// SIMATIC STEP 7 (V5.x) project Post-Platform V2
// CPU: CPU 313
// CPU: CPU 312IFM
// station: Hardware
// station: Master
// station: Hardware
// station: Slave
// station: P_ADR_BUS
// station: P_ADR_BUS
// station: P_ADR_BUS
// station: Configuration
// program: S7 Program(1)
// program: S7 Program(2)

SYMBOL_TABLE
"Counter.Balk"	C 0	COUNTER
"Geheugen.Platform"	DB 1	DB 1
"Geheugen.Instellingen"	DB 2	DB 2
"Uitgangen.Sturen"	FC 1	FC 1
"Merkers.Sturen"	FC 2	FC 2
"Timers + Counters"	FC 3	FC 3
"Berekeningen"	FC 4	FC 4
"Grafcet"	FC 5	FC 5
"Simulatie"	FC 6	FC 6
"Watch.Dog"	FC 7	FC 7
"Sub.Basis"	FC 14	FC 14
"Sub.Keuze"	FC 15	FC 15
"Sub.Keuze.Sta.A.or.B"	FC 16	FC 16
"Stap 0.0"	M 0.0	BOOL
"Stap 0.1"	M 0.1	BOOL
"Stap 0.2"	M 0.2	BOOL
"Stap 0.3"	M 0.3	BOOL
"Stap 0.4"	M 0.4	BOOL
"Stap 0.5"	M 0.5	BOOL
"Stap 0.6"	M 0.6	BOOL
"Stap 0.7"	M 0.7	BOOL
"Stap 1.0"	M 1.0	BOOL
"Stap 1.1"	M 1.1	BOOL
"Stap 1.2"	M 1.2	BOOL
"Stap 1.3"	M 1.3	BOOL
"Stap 1.4"	M 1.4	BOOL
"Stap 1.5"	M 1.5	BOOL
"Stap 1.6"	M 1.6	BOOL
"Stap 1.7"	M 1.7	BOOL
"Stap 2.0"	M 2.0	BOOL
"Stap 2.1"	M 2.1	BOOL
"Stap 2.2"	M 2.2	BOOL
"Stap 2.3"	M 2.3	BOOL
"Stap 2.4"	M 2.4	BOOL
"Stap 2.5"	M 2.5	BOOL
"Stap 2.6"	M 2.6	BOOL
"Stap 2.7"	M 2.7	BOOL
"Stap 3.0"	M 3.0	BOOL
"Stap 3.1"	M 3.1	BOOL
"Stap 3.2"	M 3.2	BOOL
"Stap 3.3"	M 3.3	BOOL
"Stap 3.4"	M 3.4	BOOL
"Stap 3.5"	M 3.5	BOOL
"Stap 3.6"	M 3.6	BOOL
"Stap 3.7"	M 3.7	BOOL
"Stap 4.0"	M 4.0	BOOL
"Stap 4.1"	M 4.1	BOOL
"Stap 4.2"	M 4.2	BOOL
"Stap 4.3"	M 4.3	BOOL
"Stap 4.4"	M 4.4	BOOL
"Stap 4.5"	M 4.5	BOOL
"Stap 4.6"	M 4.6	BOOL
"Stap 4.7"	M 4.7	BOOL
"Stop.Hardware"	M 10.0	BOOL
"Start.Hardware"	M 10.1	BOOL
"Sens.Sta.A.In"	M 10.2	BOOL
"Sens.Sta.A.Forward"	M 10.3	BOOL
"Sens.Sta.A.Down"	M 10.4	BOOL
"Sens.Sta.A.Up"	M 10.5	BOOL
"Sens.Sta.B.In"	M 10.6	BOOL
"Sens.Sta.B.Forward"	M 10.7	BOOL
"Sens.Sta.B.Down"	M 11.0	BOOL
"Sens.Sta.B.Up"	M 11.1	BOOL
"Sens.Proxi.1"	M 11.2	BOOL
"Sens.Proxi.2"	M 11.3	BOOL
"NoodStop.Relais"	M 11.4	BOOL
"Leeg"	M 12.0	BOOL
"Motor.Platform.Rechts"	M 12.1	BOOL
"Station.A.Down"	M 12.2	BOOL
"Station.A.Forward"	M 12.3	BOOL
"Station.B.Down"	M 12.4	BOOL
"Station.B.In"	M 12.5	BOOL
"Sign.Rood"	M 12.6	BOOL
"Sign.Groen"	M 12.7	BOOL
"Motor.Platform.Links"	M 13.0	BOOL
"Opstart.Cycle"	M 14.0	BOOL
"Sim.start"	M 14.1	BOOL
"Sim.Reset"	M 14.2	BOOL
"Restart"	M 14.3	BOOL
"Stop.Cycle"	M 14.4	BOOL
"Restart.Cycle"	M 14.5	BOOL
"Blinker.4s"	M 100.4	BOOL
"Blinker.5s"	M 100.5	BOOL
"Blinker.6s"	M 100.6	BOOL
"Restart.OB100"	M 101.0	BOOL
"Ingangen I0.x"	MB 10	BYTE
"Ingangen I124.x"	MB 11	BYTE
"Uitgangen Q0.x"	MB 12	BYTE
"Uitgangen Q124.x"	MB 13	BYTE
"Blinkers"	MB 100	BYTE
"Programma.Cyclus"	OB 1	OB 1
"COMPLETE RESTART"	OB 100	OB 100	// Complete Restart
"Motor.Check"	T 0	TIMER
"Platform.Vertraging"	T 1	TIMER
END_SYMBOL_TABLE

FUNCTION "Uitgangen.Sturen" : VOID	// FC 1
VERSION : 0.1
BEGIN
// (block stored without names or comments; labels and parameter names are numbered)
END_FUNCTION

FUNCTION "Merkers.Sturen" : VOID	// FC 2
VERSION : 0.1
BEGIN
// (block stored without names or comments; labels and parameter names are numbered)
END_FUNCTION

FUNCTION "Timers + Counters" : VOID	// FC 3
VERSION : 0.1
VAR_TEMP
  C0WaardeBCD : WORD ;
END_VAR
BEGIN
NETWORK
TITLE = Counter.Balk
      A     "Stap 1.2";
      CU    "Counter.Balk";
      NOP   0;
      NOP   0;
      NOP   0;
      NOP   0;
      NOP   0;
      LC    "Counter.Balk";
      T     #C0WaardeBCD;
      NOP   0;
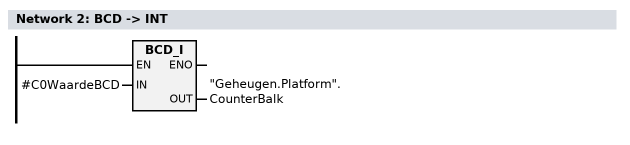
NETWORK
TITLE = BCD -> INT
      L     #C0WaardeBCD;
      BTI;
      T     "Geheugen.Platform".CounterBalk;
      NOP   0;
END_FUNCTION

FUNCTION "Berekeningen" : VOID	// FC 4
VERSION : 0.1
BEGIN
// (block stored without names or comments; labels and parameter names are numbered)
END_FUNCTION

FUNCTION "Grafcet" : VOID	// FC 5
TITLE = Grafcet
VERSION : 0.1
BEGIN
NETWORK
TITLE = Opstart
//*********************************************//
// Function: Opstart Procédure                 //
//*********************************************//
      NOP   0;
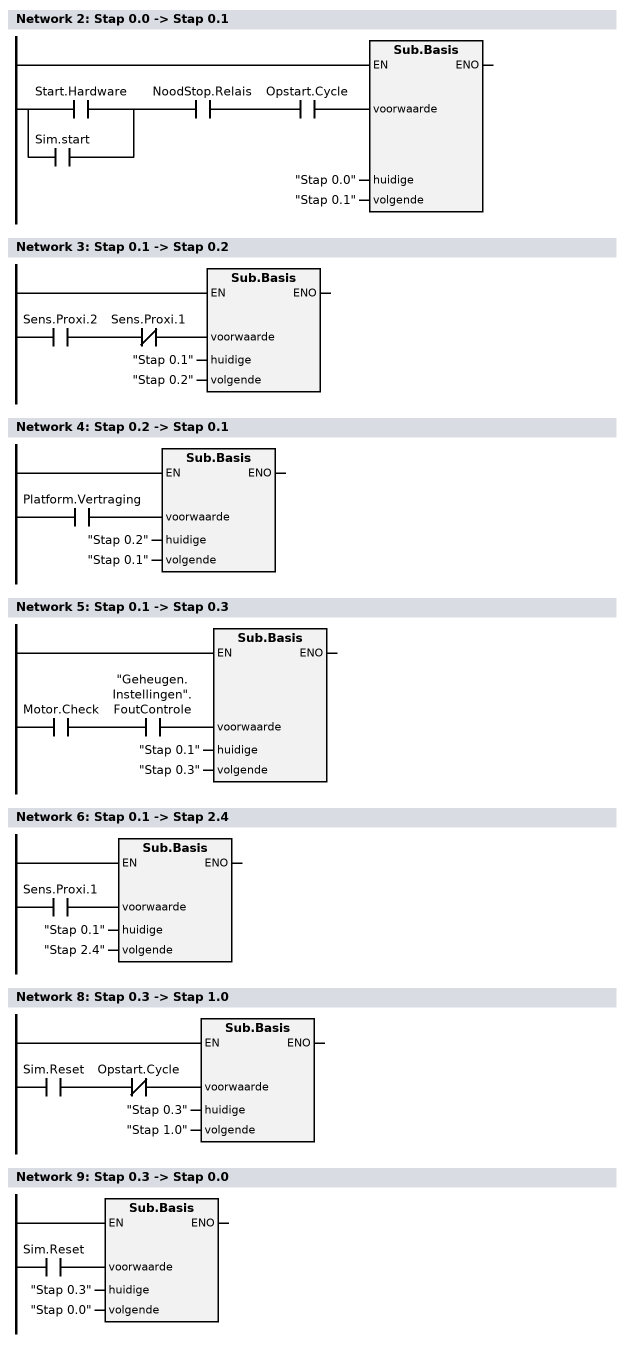
NETWORK
TITLE = Stap 0.0 -> Stap 0.1
      A(;
      O     "Start.Hardware";
      O     "Sim.start";
      );
      A     "NoodStop.Relais";
      A     "Opstart.Cycle";
      =     L 0.0;
      BLD   103;
      CALL  "Sub.Basis" (
           voorwaarde               := L 0.0,
           huidige                  := "Stap 0.0",
           volgende                 := "Stap 0.1");
      NOP   0;
NETWORK
TITLE = Stap 0.1 -> Stap 0.2
      A     "Sens.Proxi.2";
      AN    "Sens.Proxi.1";
      =     L 0.0;
      BLD   103;
      CALL  "Sub.Basis" (
           voorwaarde               := L 0.0,
           huidige                  := "Stap 0.1",
           volgende                 := "Stap 0.2");
      NOP   0;
NETWORK
TITLE = Stap 0.2 -> Stap 0.1
      A     "Platform.Vertraging";
      =     L 0.0;
      BLD   103;
      CALL  "Sub.Basis" (
           voorwaarde               := L 0.0,
           huidige                  := "Stap 0.2",
           volgende                 := "Stap 0.1");
      NOP   0;
NETWORK
TITLE = Stap 0.1 -> Stap 0.3
      A     "Motor.Check";
      A     "Geheugen.Instellingen".FoutControle;
      =     L 0.0;
      BLD   103;
      CALL  "Sub.Basis" (
           voorwaarde               := L 0.0,
           huidige                  := "Stap 0.1",
           volgende                 := "Stap 0.3");
      NOP   0;
NETWORK
TITLE = Stap 0.1 -> Stap 2.4
      A     "Sens.Proxi.1";
      =     L 0.0;
      BLD   103;
      CALL  "Sub.Basis" (
           voorwaarde               := L 0.0,
           huidige                  := "Stap 0.1",
           volgende                 := "Stap 2.4");
      NOP   0;
NETWORK
TITLE =
//*********************************************//
// Function: Einde Opstart Procédure           //
//           Begin Fout Procédure              //
//*********************************************//
      NOP   0;
NETWORK
TITLE = Stap 0.3 -> Stap 1.0
      A     "Sim.Reset";
      AN    "Opstart.Cycle";
      =     L 0.0;
      BLD   103;
      CALL  "Sub.Basis" (
           voorwaarde               := L 0.0,
           huidige                  := "Stap 0.3",
           volgende                 := "Stap 1.0");
      NOP   0;
NETWORK
TITLE = Stap 0.3 -> Stap 0.0
//Fout motor platform
      A     "Sim.Reset";
      =     L 0.0;
      BLD   103;
      CALL  "Sub.Basis" (
           voorwaarde               := L 0.0,
           huidige                  := "Stap 0.3",
           volgende                 := "Stap 0.0");
      NOP   0;
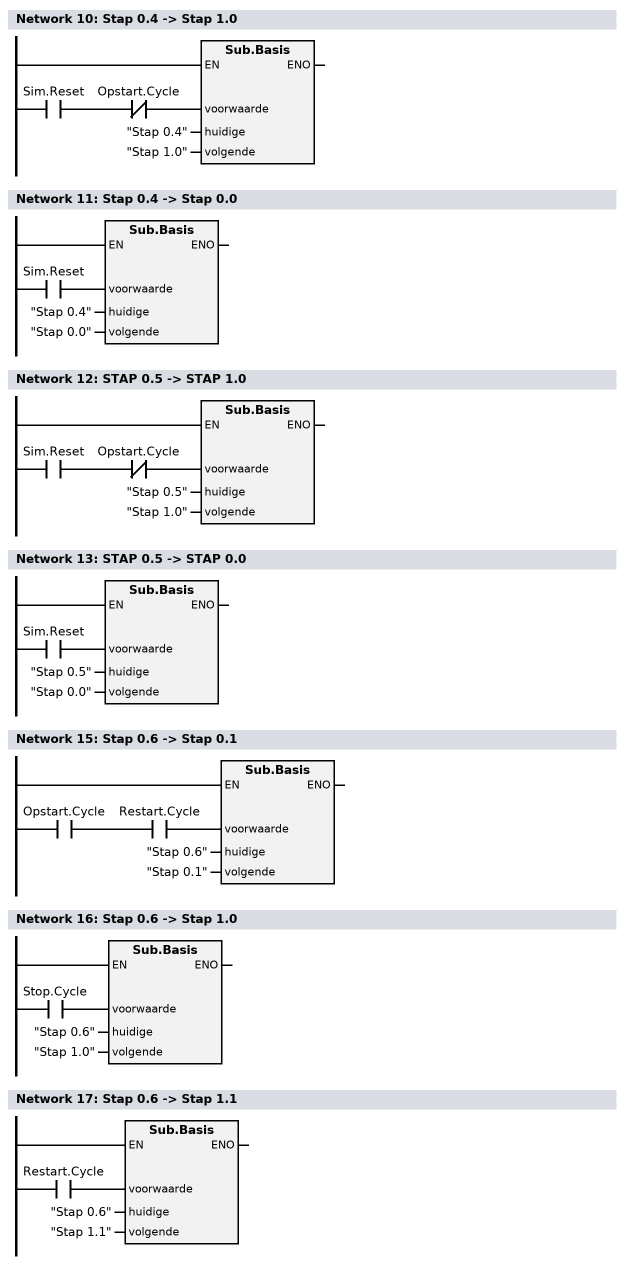
NETWORK
TITLE = Stap 0.4 -> Stap 1.0
//Fout Station A
//
      A     "Sim.Reset";
      AN    "Opstart.Cycle";
      =     L 0.0;
      BLD   103;
      CALL  "Sub.Basis" (
           voorwaarde               := L 0.0,
           huidige                  := "Stap 0.4",
           volgende                 := "Stap 1.0");
      NOP   0;
NETWORK
TITLE = Stap 0.4 -> Stap 0.0
//Fout Station A
      A     "Sim.Reset";
      =     L 0.0;
      BLD   103;
      CALL  "Sub.Basis" (
           voorwaarde               := L 0.0,
           huidige                  := "Stap 0.4",
           volgende                 := "Stap 0.0");
      NOP   0;
NETWORK
TITLE = STAP 0.5 -> STAP 1.0
//FOUT STATION B
      A     "Sim.Reset";
      AN    "Opstart.Cycle";
      =     L 0.0;
      BLD   103;
      CALL  "Sub.Basis" (
           voorwaarde               := L 0.0,
           huidige                  := "Stap 0.5",
           volgende                 := "Stap 1.0");
      NOP   0;
NETWORK
TITLE = STAP 0.5 -> STAP 0.0
//FOUT STATION B
      A     "Sim.Reset";
      =     L 0.0;
      BLD   103;
      CALL  "Sub.Basis" (
           voorwaarde               := L 0.0,
           huidige                  := "Stap 0.5",
           volgende                 := "Stap 0.0");
      NOP   0;
NETWORK
TITLE =
//*********************************************//
// Function: Einde FOUT Procédur               //
//           Begin STOP Procédure              //
//*********************************************//
      NOP   0;
NETWORK
TITLE = Stap 0.6 -> Stap 0.1
//Machine onderbroken door stop
//
      A     "Opstart.Cycle";
      A     "Restart.Cycle";
      =     L 0.0;
      BLD   103;
      CALL  "Sub.Basis" (
           voorwaarde               := L 0.0,
           huidige                  := "Stap 0.6",
           volgende                 := "Stap 0.1");
      NOP   0;
NETWORK
TITLE = Stap 0.6 -> Stap 1.0
//Machine onderbroken door stop
//
      A     "Stop.Cycle";
      =     L 0.0;
      BLD   103;
      CALL  "Sub.Basis" (
           voorwaarde               := L 0.0,
           huidige                  := "Stap 0.6",
           volgende                 := "Stap 1.0");
      NOP   0;
NETWORK
TITLE = Stap 0.6 -> Stap 1.1
//Machine onderbroken door stop
//
      A     "Restart.Cycle";
      =     L 0.0;
      BLD   103;
      CALL  "Sub.Basis" (
           voorwaarde               := L 0.0,
           huidige                  := "Stap 0.6",
           volgende                 := "Stap 1.1");
      NOP   0;
NETWORK
TITLE =
//*********************************************//
// Function: Einde STOP Procédur               //
//           Begin Normale Procédure           //
//*********************************************//
      NOP   0;
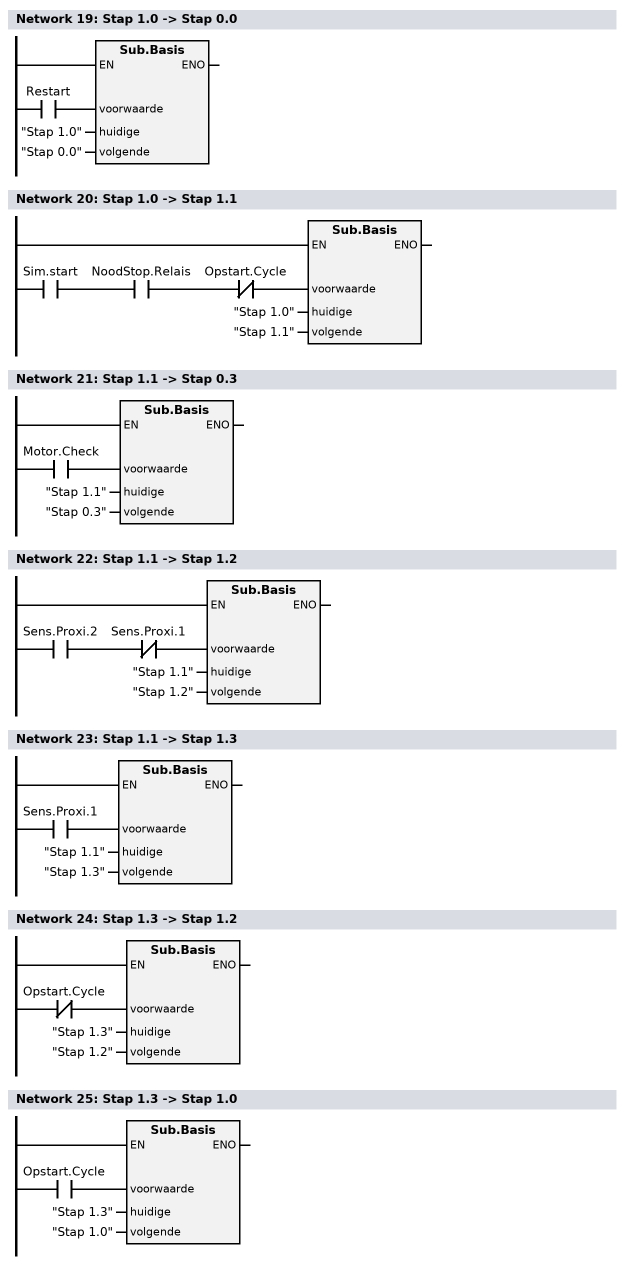
NETWORK
TITLE = Stap 1.0 -> Stap 0.0
      A     "Restart";
      =     L 0.0;
      BLD   103;
      CALL  "Sub.Basis" (
           voorwaarde               := L 0.0,
           huidige                  := "Stap 1.0",
           volgende                 := "Stap 0.0");
      NOP   0;
NETWORK
TITLE = Stap 1.0 -> Stap 1.1
      A     "Sim.start";
      A     "NoodStop.Relais";
      AN    "Opstart.Cycle";
      =     L 0.0;
      BLD   103;
      CALL  "Sub.Basis" (
           voorwaarde               := L 0.0,
           huidige                  := "Stap 1.0",
           volgende                 := "Stap 1.1");
      NOP   0;
NETWORK
TITLE = Stap 1.1 -> Stap 0.3
      A     "Motor.Check";
      =     L 0.0;
      BLD   103;
      CALL  "Sub.Basis" (
           voorwaarde               := L 0.0,
           huidige                  := "Stap 1.1",
           volgende                 := "Stap 0.3");
      NOP   0;
NETWORK
TITLE = Stap 1.1 -> Stap 1.2
      A     "Sens.Proxi.2";
      AN    "Sens.Proxi.1";
      =     L 0.0;
      BLD   103;
      CALL  "Sub.Basis" (
           voorwaarde               := L 0.0,
           huidige                  := "Stap 1.1",
           volgende                 := "Stap 1.2");
      NOP   0;
NETWORK
TITLE = Stap 1.1 -> Stap 1.3
      A     "Sens.Proxi.1";
      =     L 0.0;
      BLD   103;
      CALL  "Sub.Basis" (
           voorwaarde               := L 0.0,
           huidige                  := "Stap 1.1",
           volgende                 := "Stap 1.3");
      NOP   0;
NETWORK
TITLE = Stap 1.3 -> Stap 1.2
      AN    "Opstart.Cycle";
      =     L 0.0;
      BLD   103;
      CALL  "Sub.Basis" (
           voorwaarde               := L 0.0,
           huidige                  := "Stap 1.3",
           volgende                 := "Stap 1.2");
      NOP   0;
NETWORK
TITLE = Stap 1.3 -> Stap 1.0
      A     "Opstart.Cycle";
      =     L 0.0;
      BLD   103;
      CALL  "Sub.Basis" (
           voorwaarde               := L 0.0,
           huidige                  := "Stap 1.3",
           volgende                 := "Stap 1.0");
      NOP   0;
NETWORK
TITLE =
//*********************************************//
// Function: Einde Normale Procédure           //
//           Begin Kies Procédure              //
//*********************************************//
      NOP   0;
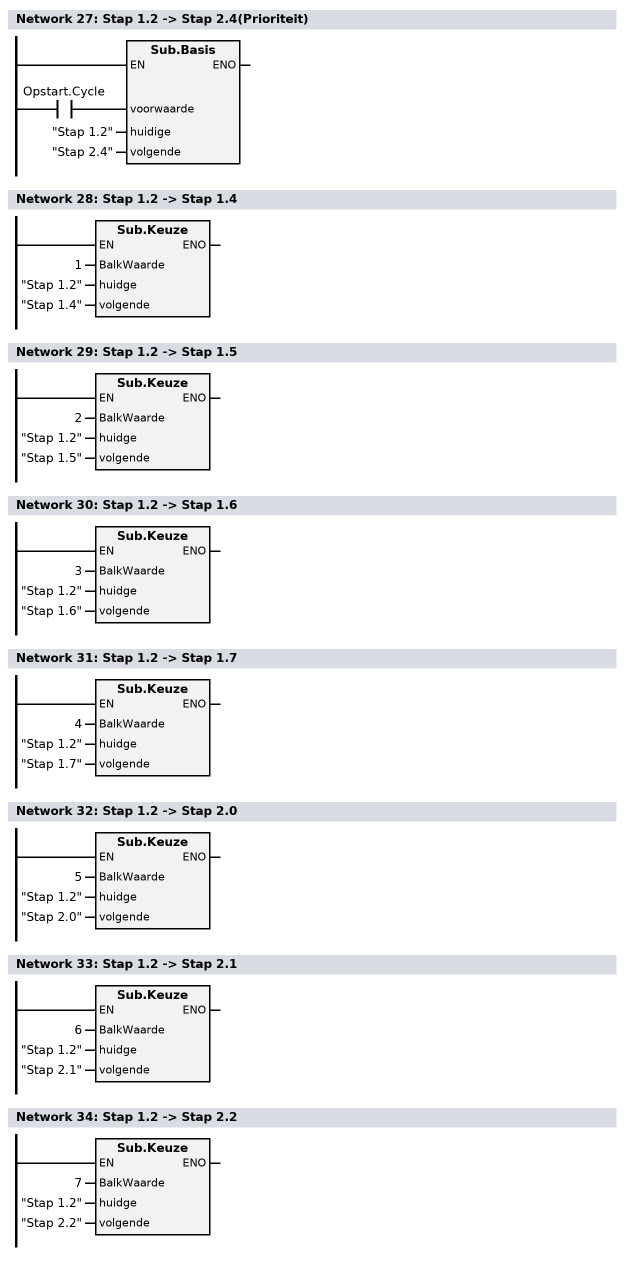
NETWORK
TITLE = Stap 1.2 -> Stap 2.4(Prioriteit)
      A     "Opstart.Cycle";
      =     L 0.0;
      BLD   103;
      CALL  "Sub.Basis" (
           voorwaarde               := L 0.0,
           huidige                  := "Stap 1.2",
           volgende                 := "Stap 2.4");
      NOP   0;
NETWORK
TITLE = Stap 1.2 -> Stap 1.4
      CALL  "Sub.Keuze" (
           BalkWaarde               := 1,
           huidge                   := "Stap 1.2",
           volgende                 := "Stap 1.4");
      NOP   0;
NETWORK
TITLE = Stap 1.2 -> Stap 1.5
      CALL  "Sub.Keuze" (
           BalkWaarde               := 2,
           huidge                   := "Stap 1.2",
           volgende                 := "Stap 1.5");
      NOP   0;
NETWORK
TITLE = Stap 1.2 -> Stap 1.6
      CALL  "Sub.Keuze" (
           BalkWaarde               := 3,
           huidge                   := "Stap 1.2",
           volgende                 := "Stap 1.6");
      NOP   0;
NETWORK
TITLE = Stap 1.2 -> Stap 1.7
      CALL  "Sub.Keuze" (
           BalkWaarde               := 4,
           huidge                   := "Stap 1.2",
           volgende                 := "Stap 1.7");
      NOP   0;
NETWORK
TITLE = Stap 1.2 -> Stap 2.0
      CALL  "Sub.Keuze" (
           BalkWaarde               := 5,
           huidge                   := "Stap 1.2",
           volgende                 := "Stap 2.0");
      NOP   0;
NETWORK
TITLE = Stap 1.2 -> Stap 2.1
      CALL  "Sub.Keuze" (
           BalkWaarde               := 6,
           huidge                   := "Stap 1.2",
           volgende                 := "Stap 2.1");
      NOP   0;
NETWORK
TITLE = Stap 1.2 -> Stap 2.2
      CALL  "Sub.Keuze" (
           BalkWaarde               := 7,
           huidge                   := "Stap 1.2",
           volgende                 := "Stap 2.2");
      NOP   0;
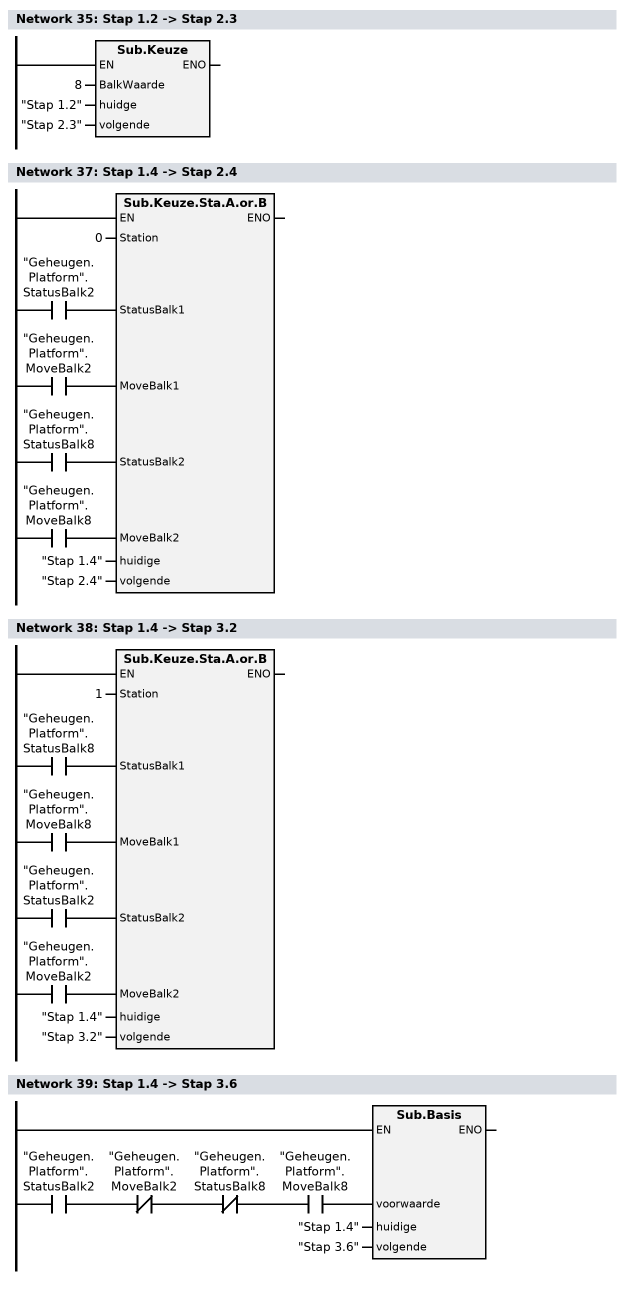
NETWORK
TITLE = Stap 1.2 -> Stap 2.3
      CALL  "Sub.Keuze" (
           BalkWaarde               := 8,
           huidge                   := "Stap 1.2",
           volgende                 := "Stap 2.3");
      NOP   0;
NETWORK
TITLE =
//*********************************************//
// Function: Einde Kies Procédure              //
//           Begin Station Keuze Procédure     //
//           Waarde Counter CO: 1              //
//*********************************************//
      NOP   0;
NETWORK
TITLE = Stap 1.4 -> Stap 2.4
//Naar Station A
      A     "Geheugen.Platform".StatusBalk2;
      =     L 0.0;
      BLD   103;
      A     "Geheugen.Platform".MoveBalk2;
      =     L 0.1;
      BLD   103;
      A     "Geheugen.Platform".StatusBalk8;
      =     L 0.2;
      BLD   103;
      A     "Geheugen.Platform".MoveBalk8;
      =     L 0.3;
      BLD   103;
      CALL  "Sub.Keuze.Sta.A.or.B" (
           Station                  := 0,
           StatusBalk1              := L 0.0,
           MoveBalk1                := L 0.1,
           StatusBalk2              := L 0.2,
           MoveBalk2                := L 0.3,
           huidige                  := "Stap 1.4",
           volgende                 := "Stap 2.4");
      NOP   0;
NETWORK
TITLE = Stap 1.4 -> Stap 3.2
//Naar Station B
      A     "Geheugen.Platform".StatusBalk8;
      =     L 0.0;
      BLD   103;
      A     "Geheugen.Platform".MoveBalk8;
      =     L 0.1;
      BLD   103;
      A     "Geheugen.Platform".StatusBalk2;
      =     L 0.2;
      BLD   103;
      A     "Geheugen.Platform".MoveBalk2;
      =     L 0.3;
      BLD   103;
      CALL  "Sub.Keuze.Sta.A.or.B" (
           Station                  := 1,
           StatusBalk1              := L 0.0,
           MoveBalk1                := L 0.1,
           StatusBalk2              := L 0.2,
           MoveBalk2                := L 0.3,
           huidige                  := "Stap 1.4",
           volgende                 := "Stap 3.2");
      NOP   0;
NETWORK
TITLE = Stap 1.4 -> Stap 3.6
//Station A + B
      A     "Geheugen.Platform".StatusBalk2;
      AN    "Geheugen.Platform".MoveBalk2;
      AN    "Geheugen.Platform".StatusBalk8;
      A     "Geheugen.Platform".MoveBalk8;
      =     L 0.0;
      BLD   103;
      CALL  "Sub.Basis" (
           voorwaarde               := L 0.0,
           huidige                  := "Stap 1.4",
           volgende                 := "Stap 3.6");
      NOP   0;
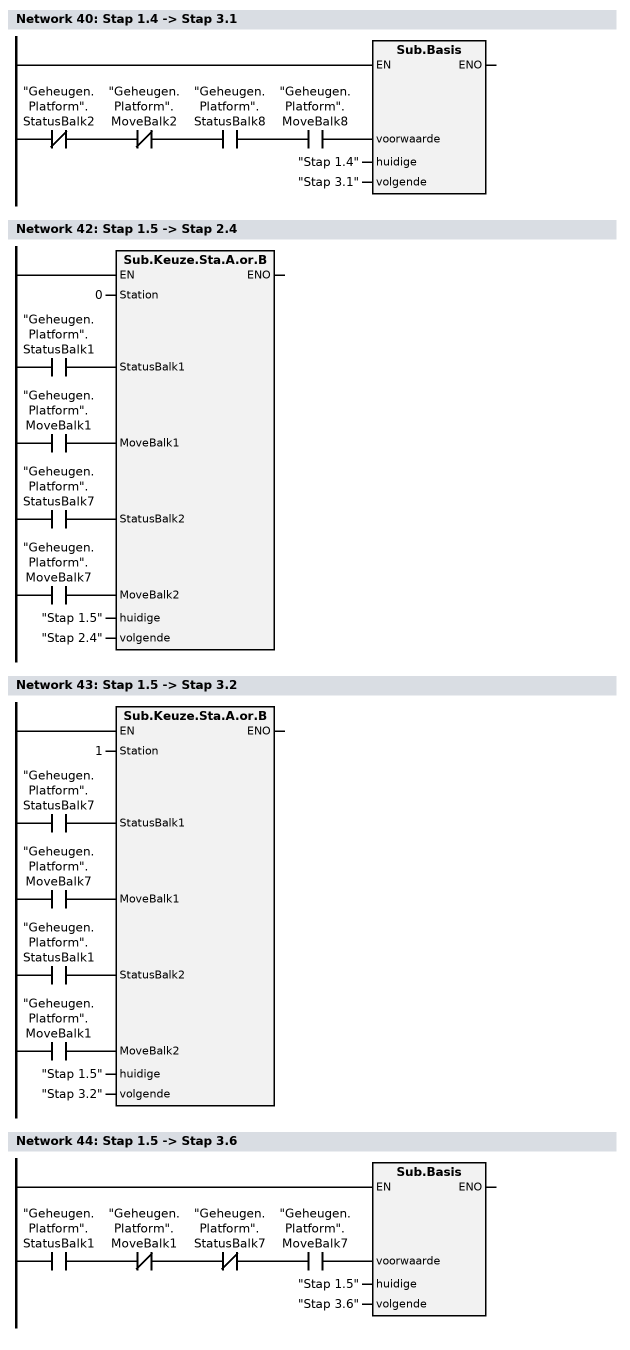
NETWORK
TITLE = Stap 1.4 -> Stap 3.1
//Geen actie
//
      AN    "Geheugen.Platform".StatusBalk2;
      AN    "Geheugen.Platform".MoveBalk2;
      A     "Geheugen.Platform".StatusBalk8;
      A     "Geheugen.Platform".MoveBalk8;
      =     L 0.0;
      BLD   103;
      CALL  "Sub.Basis" (
           voorwaarde               := L 0.0,
           huidige                  := "Stap 1.4",
           volgende                 := "Stap 3.1");
      NOP   0;
NETWORK
TITLE =
//*********************************************//
// Function: Einde Waarde Counter CO: 1        //
//           Begin Waarde Counter CO: 2        //
//*********************************************//
      NOP   0;
NETWORK
TITLE = Stap 1.5 -> Stap 2.4
//Naar Station A
      A     "Geheugen.Platform".StatusBalk1;
      =     L 0.0;
      BLD   103;
      A     "Geheugen.Platform".MoveBalk1;
      =     L 0.1;
      BLD   103;
      A     "Geheugen.Platform".StatusBalk7;
      =     L 0.2;
      BLD   103;
      A     "Geheugen.Platform".MoveBalk7;
      =     L 0.3;
      BLD   103;
      CALL  "Sub.Keuze.Sta.A.or.B" (
           Station                  := 0,
           StatusBalk1              := L 0.0,
           MoveBalk1                := L 0.1,
           StatusBalk2              := L 0.2,
           MoveBalk2                := L 0.3,
           huidige                  := "Stap 1.5",
           volgende                 := "Stap 2.4");
      NOP   0;
NETWORK
TITLE = Stap 1.5 -> Stap 3.2
//Naar Station B
      A     "Geheugen.Platform".StatusBalk7;
      =     L 0.0;
      BLD   103;
      A     "Geheugen.Platform".MoveBalk7;
      =     L 0.1;
      BLD   103;
      A     "Geheugen.Platform".StatusBalk1;
      =     L 0.2;
      BLD   103;
      A     "Geheugen.Platform".MoveBalk1;
      =     L 0.3;
      BLD   103;
      CALL  "Sub.Keuze.Sta.A.or.B" (
           Station                  := 1,
           StatusBalk1              := L 0.0,
           MoveBalk1                := L 0.1,
           StatusBalk2              := L 0.2,
           MoveBalk2                := L 0.3,
           huidige                  := "Stap 1.5",
           volgende                 := "Stap 3.2");
      NOP   0;
NETWORK
TITLE = Stap 1.5 -> Stap 3.6
//Station A + B
      A     "Geheugen.Platform".StatusBalk1;
      AN    "Geheugen.Platform".MoveBalk1;
      AN    "Geheugen.Platform".StatusBalk7;
      A     "Geheugen.Platform".MoveBalk7;
      =     L 0.0;
      BLD   103;
      CALL  "Sub.Basis" (
           voorwaarde               := L 0.0,
           huidige                  := "Stap 1.5",
           volgende                 := "Stap 3.6");
      NOP   0;
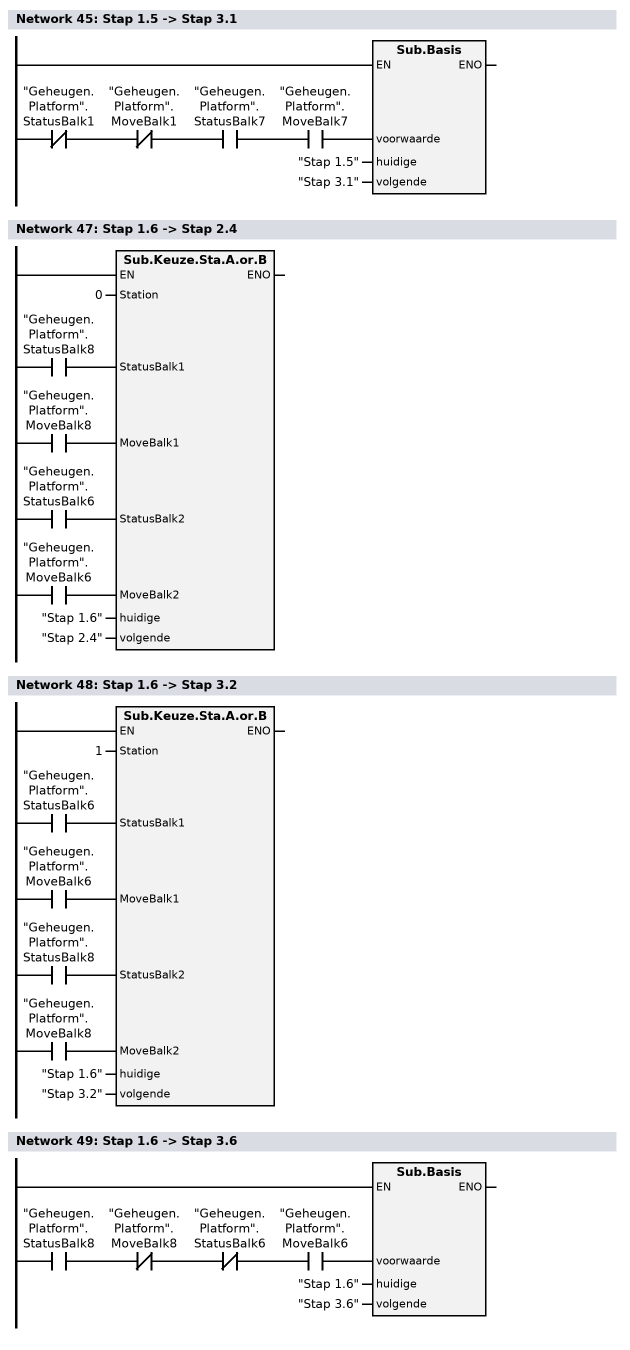
NETWORK
TITLE = Stap 1.5 -> Stap 3.1
//Geen actie
//
      AN    "Geheugen.Platform".StatusBalk1;
      AN    "Geheugen.Platform".MoveBalk1;
      A     "Geheugen.Platform".StatusBalk7;
      A     "Geheugen.Platform".MoveBalk7;
      =     L 0.0;
      BLD   103;
      CALL  "Sub.Basis" (
           voorwaarde               := L 0.0,
           huidige                  := "Stap 1.5",
           volgende                 := "Stap 3.1");
      NOP   0;
NETWORK
TITLE =
//*********************************************//
// Function: Einde Waarde Counter CO: 2        //
//           Begin Waarde Counter CO: 3        //
//*********************************************//
      NOP   0;
NETWORK
TITLE = Stap 1.6 -> Stap 2.4
//Naar Station A
      A     "Geheugen.Platform".StatusBalk8;
      =     L 0.0;
      BLD   103;
      A     "Geheugen.Platform".MoveBalk8;
      =     L 0.1;
      BLD   103;
      A     "Geheugen.Platform".StatusBalk6;
      =     L 0.2;
      BLD   103;
      A     "Geheugen.Platform".MoveBalk6;
      =     L 0.3;
      BLD   103;
      CALL  "Sub.Keuze.Sta.A.or.B" (
           Station                  := 0,
           StatusBalk1              := L 0.0,
           MoveBalk1                := L 0.1,
           StatusBalk2              := L 0.2,
           MoveBalk2                := L 0.3,
           huidige                  := "Stap 1.6",
           volgende                 := "Stap 2.4");
      NOP   0;
NETWORK
TITLE = Stap 1.6 -> Stap 3.2
//Naar Station B
      A     "Geheugen.Platform".StatusBalk6;
      =     L 0.0;
      BLD   103;
      A     "Geheugen.Platform".MoveBalk6;
      =     L 0.1;
      BLD   103;
      A     "Geheugen.Platform".StatusBalk8;
      =     L 0.2;
      BLD   103;
      A     "Geheugen.Platform".MoveBalk8;
      =     L 0.3;
      BLD   103;
      CALL  "Sub.Keuze.Sta.A.or.B" (
           Station                  := 1,
           StatusBalk1              := L 0.0,
           MoveBalk1                := L 0.1,
           StatusBalk2              := L 0.2,
           MoveBalk2                := L 0.3,
           huidige                  := "Stap 1.6",
           volgende                 := "Stap 3.2");
      NOP   0;
NETWORK
TITLE = Stap 1.6 -> Stap 3.6
//Station A + B
      A     "Geheugen.Platform".StatusBalk8;
      AN    "Geheugen.Platform".MoveBalk8;
      AN    "Geheugen.Platform".StatusBalk6;
      A     "Geheugen.Platform".MoveBalk6;
      =     L 0.0;
      BLD   103;
      CALL  "Sub.Basis" (
           voorwaarde               := L 0.0,
           huidige                  := "Stap 1.6",
           volgende                 := "Stap 3.6");
      NOP   0;
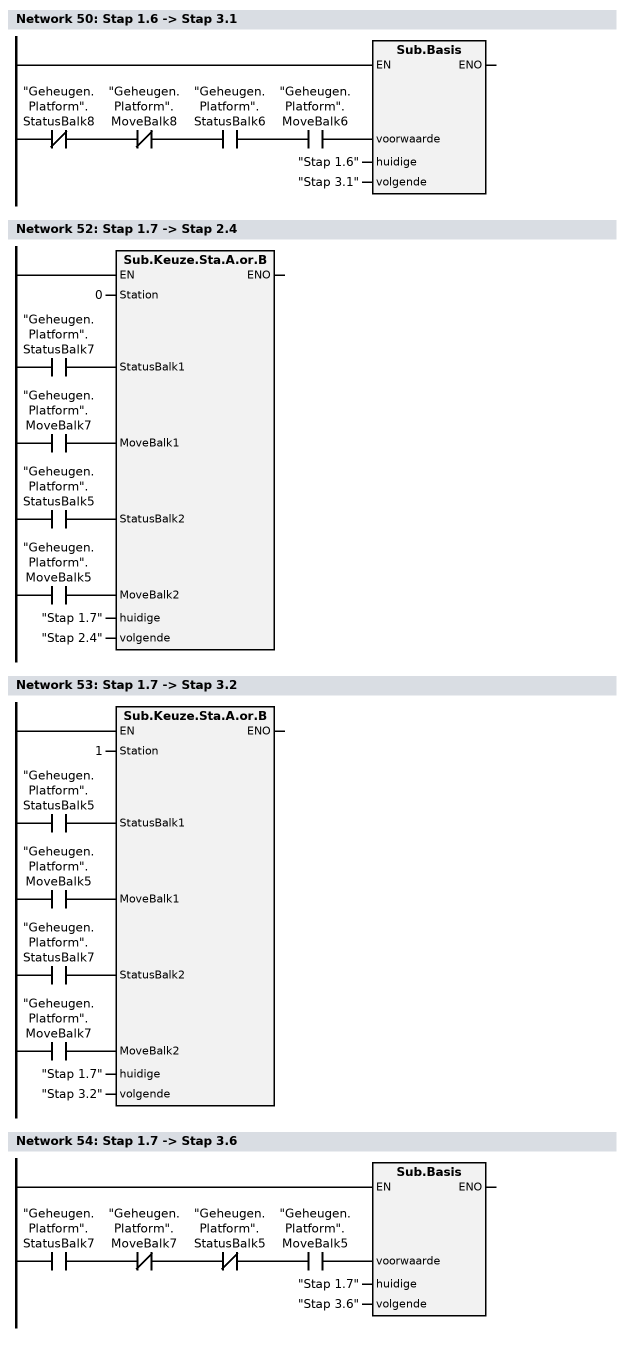
NETWORK
TITLE = Stap 1.6 -> Stap 3.1
//Geen actie
//
      AN    "Geheugen.Platform".StatusBalk8;
      AN    "Geheugen.Platform".MoveBalk8;
      A     "Geheugen.Platform".StatusBalk6;
      A     "Geheugen.Platform".MoveBalk6;
      =     L 0.0;
      BLD   103;
      CALL  "Sub.Basis" (
           voorwaarde               := L 0.0,
           huidige                  := "Stap 1.6",
           volgende                 := "Stap 3.1");
      NOP   0;
NETWORK
TITLE =
//*********************************************//
// Function: Einde Waarde Counter CO: 3        //
//           Begin Waarde Counter CO: 4        //
//*********************************************//
      NOP   0;
NETWORK
TITLE = Stap 1.7 -> Stap 2.4
//Naar Station A
      A     "Geheugen.Platform".StatusBalk7;
      =     L 0.0;
      BLD   103;
      A     "Geheugen.Platform".MoveBalk7;
      =     L 0.1;
      BLD   103;
      A     "Geheugen.Platform".StatusBalk5;
      =     L 0.2;
      BLD   103;
      A     "Geheugen.Platform".MoveBalk5;
      =     L 0.3;
      BLD   103;
      CALL  "Sub.Keuze.Sta.A.or.B" (
           Station                  := 0,
           StatusBalk1              := L 0.0,
           MoveBalk1                := L 0.1,
           StatusBalk2              := L 0.2,
           MoveBalk2                := L 0.3,
           huidige                  := "Stap 1.7",
           volgende                 := "Stap 2.4");
      NOP   0;
NETWORK
TITLE = Stap 1.7 -> Stap 3.2
//Naar Station B
      A     "Geheugen.Platform".StatusBalk5;
      =     L 0.0;
      BLD   103;
      A     "Geheugen.Platform".MoveBalk5;
      =     L 0.1;
      BLD   103;
      A     "Geheugen.Platform".StatusBalk7;
      =     L 0.2;
      BLD   103;
      A     "Geheugen.Platform".MoveBalk7;
      =     L 0.3;
      BLD   103;
      CALL  "Sub.Keuze.Sta.A.or.B" (
           Station                  := 1,
           StatusBalk1              := L 0.0,
           MoveBalk1                := L 0.1,
           StatusBalk2              := L 0.2,
           MoveBalk2                := L 0.3,
           huidige                  := "Stap 1.7",
           volgende                 := "Stap 3.2");
      NOP   0;
NETWORK
TITLE = Stap 1.7 -> Stap 3.6
//Station A + B
      A     "Geheugen.Platform".StatusBalk7;
      AN    "Geheugen.Platform".MoveBalk7;
      AN    "Geheugen.Platform".StatusBalk5;
      A     "Geheugen.Platform".MoveBalk5;
      =     L 0.0;
      BLD   103;
      CALL  "Sub.Basis" (
           voorwaarde               := L 0.0,
           huidige                  := "Stap 1.7",
           volgende                 := "Stap 3.6");
      NOP   0;
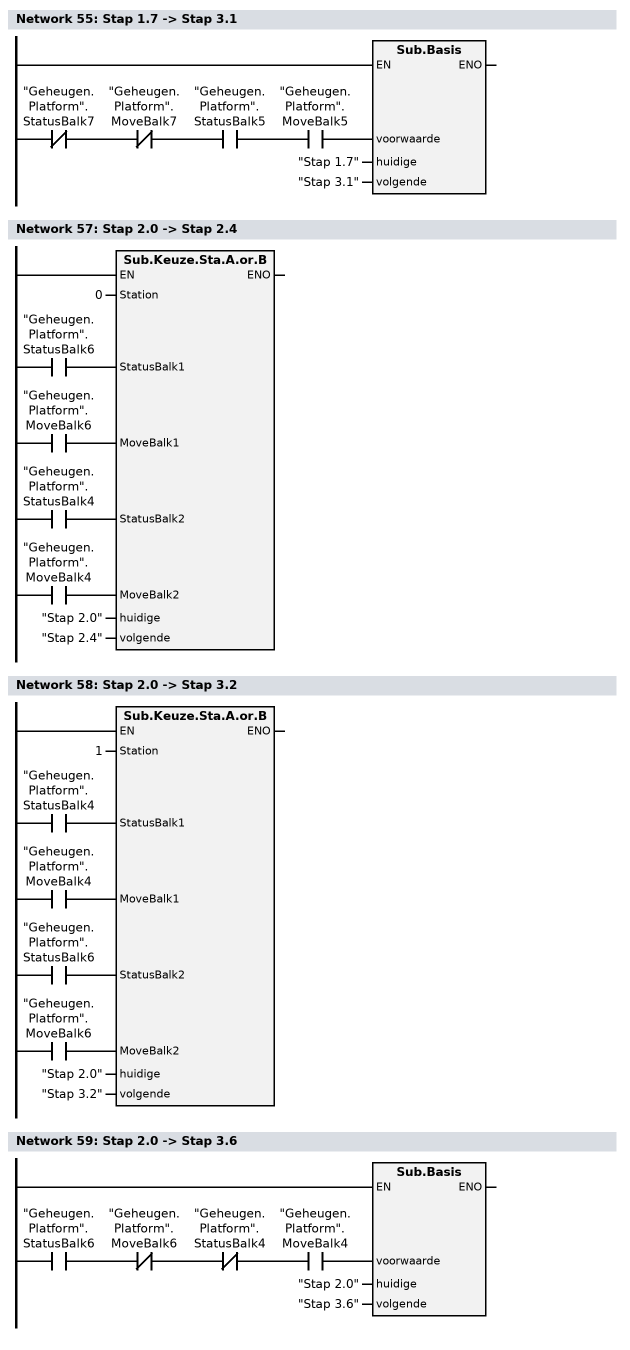
NETWORK
TITLE = Stap 1.7 -> Stap 3.1
//Geen actie
//
      AN    "Geheugen.Platform".StatusBalk7;
      AN    "Geheugen.Platform".MoveBalk7;
      A     "Geheugen.Platform".StatusBalk5;
      A     "Geheugen.Platform".MoveBalk5;
      =     L 0.0;
      BLD   103;
      CALL  "Sub.Basis" (
           voorwaarde               := L 0.0,
           huidige                  := "Stap 1.7",
           volgende                 := "Stap 3.1");
      NOP   0;
NETWORK
TITLE =
//*********************************************//
// Function: Einde Waarde Counter CO: 4        //
//           Begin Waarde Counter CO: 5        //
//*********************************************//
      NOP   0;
NETWORK
TITLE = Stap 2.0 -> Stap 2.4
//Naar Station A
      A     "Geheugen.Platform".StatusBalk6;
      =     L 0.0;
      BLD   103;
      A     "Geheugen.Platform".MoveBalk6;
      =     L 0.1;
      BLD   103;
      A     "Geheugen.Platform".StatusBalk4;
      =     L 0.2;
      BLD   103;
      A     "Geheugen.Platform".MoveBalk4;
      =     L 0.3;
      BLD   103;
      CALL  "Sub.Keuze.Sta.A.or.B" (
           Station                  := 0,
           StatusBalk1              := L 0.0,
           MoveBalk1                := L 0.1,
           StatusBalk2              := L 0.2,
           MoveBalk2                := L 0.3,
           huidige                  := "Stap 2.0",
           volgende                 := "Stap 2.4");
      NOP   0;
NETWORK
TITLE = Stap 2.0 -> Stap 3.2
//Naar Station B
      A     "Geheugen.Platform".StatusBalk4;
      =     L 0.0;
      BLD   103;
      A     "Geheugen.Platform".MoveBalk4;
      =     L 0.1;
      BLD   103;
      A     "Geheugen.Platform".StatusBalk6;
      =     L 0.2;
      BLD   103;
      A     "Geheugen.Platform".MoveBalk6;
      =     L 0.3;
      BLD   103;
      CALL  "Sub.Keuze.Sta.A.or.B" (
           Station                  := 1,
           StatusBalk1              := L 0.0,
           MoveBalk1                := L 0.1,
           StatusBalk2              := L 0.2,
           MoveBalk2                := L 0.3,
           huidige                  := "Stap 2.0",
           volgende                 := "Stap 3.2");
      NOP   0;
NETWORK
TITLE = Stap 2.0 -> Stap 3.6
//Station A + B
      A     "Geheugen.Platform".StatusBalk6;
      AN    "Geheugen.Platform".MoveBalk6;
      AN    "Geheugen.Platform".StatusBalk4;
      A     "Geheugen.Platform".MoveBalk4;
      =     L 0.0;
      BLD   103;
      CALL  "Sub.Basis" (
           voorwaarde               := L 0.0,
           huidige                  := "Stap 2.0",
           volgende                 := "Stap 3.6");
      NOP   0;
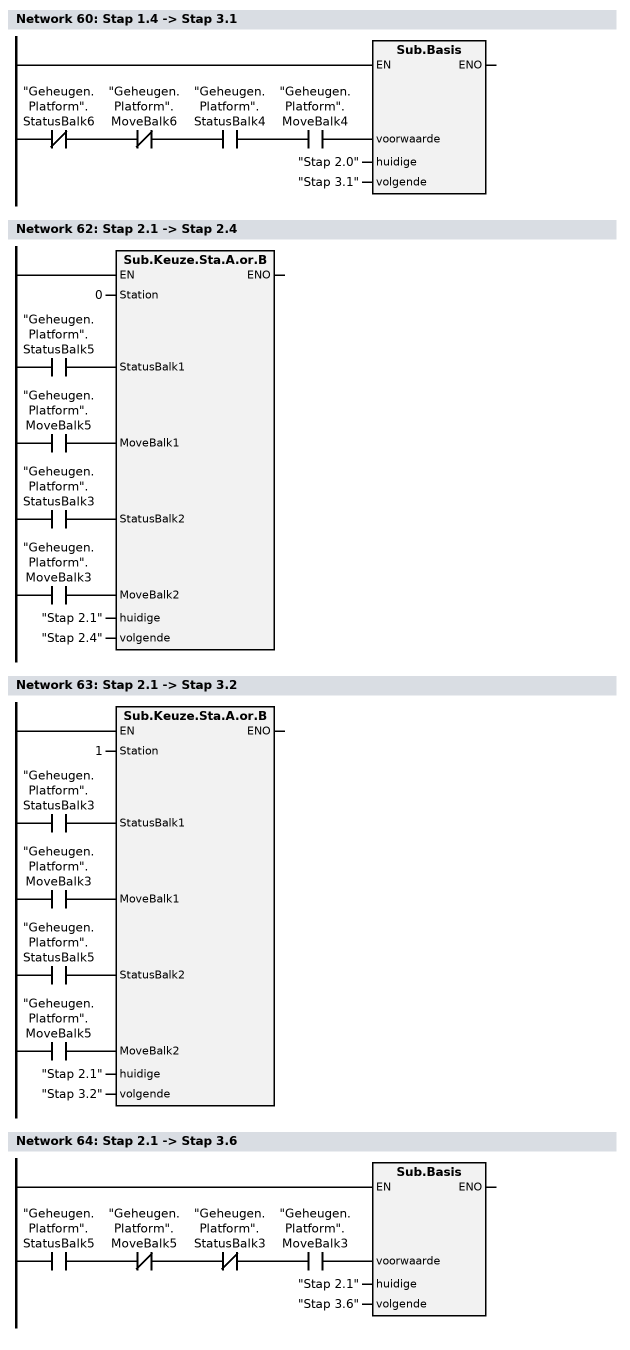
NETWORK
TITLE = Stap 1.4 -> Stap 3.1
//Geen actie
//
      AN    "Geheugen.Platform".StatusBalk6;
      AN    "Geheugen.Platform".MoveBalk6;
      A     "Geheugen.Platform".StatusBalk4;
      A     "Geheugen.Platform".MoveBalk4;
      =     L 0.0;
      BLD   103;
      CALL  "Sub.Basis" (
           voorwaarde               := L 0.0,
           huidige                  := "Stap 2.0",
           volgende                 := "Stap 3.1");
      NOP   0;
NETWORK
TITLE =
//*********************************************//
// Function: Einde Waarde Counter CO: 5        //
//           Begin Waarde Counter CO: 6        //
//*********************************************//
      NOP   0;
NETWORK
TITLE = Stap 2.1 -> Stap 2.4
//Naar Station A
      A     "Geheugen.Platform".StatusBalk5;
      =     L 0.0;
      BLD   103;
      A     "Geheugen.Platform".MoveBalk5;
      =     L 0.1;
      BLD   103;
      A     "Geheugen.Platform".StatusBalk3;
      =     L 0.2;
      BLD   103;
      A     "Geheugen.Platform".MoveBalk3;
      =     L 0.3;
      BLD   103;
      CALL  "Sub.Keuze.Sta.A.or.B" (
           Station                  := 0,
           StatusBalk1              := L 0.0,
           MoveBalk1                := L 0.1,
           StatusBalk2              := L 0.2,
           MoveBalk2                := L 0.3,
           huidige                  := "Stap 2.1",
           volgende                 := "Stap 2.4");
      NOP   0;
NETWORK
TITLE = Stap 2.1 -> Stap 3.2
//Naar Station B
      A     "Geheugen.Platform".StatusBalk3;
      =     L 0.0;
      BLD   103;
      A     "Geheugen.Platform".MoveBalk3;
      =     L 0.1;
      BLD   103;
      A     "Geheugen.Platform".StatusBalk5;
      =     L 0.2;
      BLD   103;
      A     "Geheugen.Platform".MoveBalk5;
      =     L 0.3;
      BLD   103;
      CALL  "Sub.Keuze.Sta.A.or.B" (
           Station                  := 1,
           StatusBalk1              := L 0.0,
           MoveBalk1                := L 0.1,
           StatusBalk2              := L 0.2,
           MoveBalk2                := L 0.3,
           huidige                  := "Stap 2.1",
           volgende                 := "Stap 3.2");
      NOP   0;
NETWORK
TITLE = Stap 2.1 -> Stap 3.6
//Station A + B
      A     "Geheugen.Platform".StatusBalk5;
      AN    "Geheugen.Platform".MoveBalk5;
      AN    "Geheugen.Platform".StatusBalk3;
      A     "Geheugen.Platform".MoveBalk3;
      =     L 0.0;
      BLD   103;
      CALL  "Sub.Basis" (
           voorwaarde               := L 0.0,
           huidige                  := "Stap 2.1",
           volgende                 := "Stap 3.6");
      NOP   0;
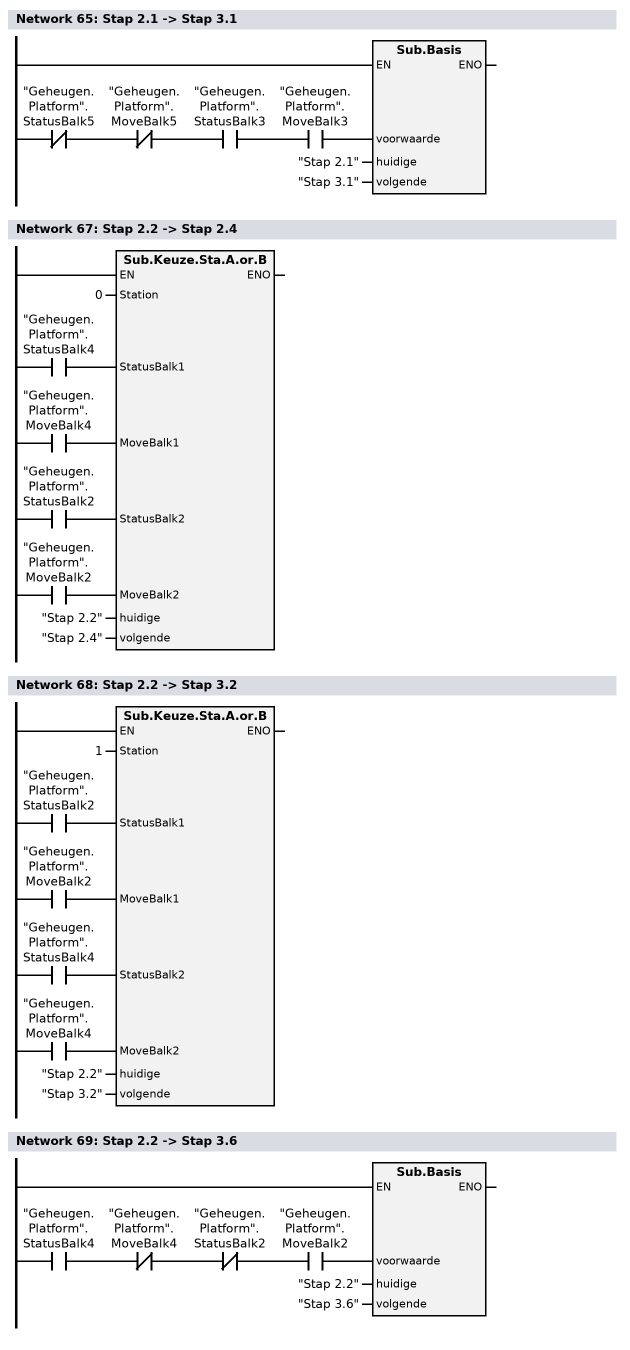
NETWORK
TITLE = Stap 2.1 -> Stap 3.1
//Geen actie
//
      AN    "Geheugen.Platform".StatusBalk5;
      AN    "Geheugen.Platform".MoveBalk5;
      A     "Geheugen.Platform".StatusBalk3;
      A     "Geheugen.Platform".MoveBalk3;
      =     L 0.0;
      BLD   103;
      CALL  "Sub.Basis" (
           voorwaarde               := L 0.0,
           huidige                  := "Stap 2.1",
           volgende                 := "Stap 3.1");
      NOP   0;
NETWORK
TITLE =
//*********************************************//
// Function: Einde Waarde Counter CO: 6        //
//           Begin Waarde Counter CO: 7        //
//*********************************************//
      NOP   0;
NETWORK
TITLE = Stap 2.2 -> Stap 2.4
//Naar Station A
      A     "Geheugen.Platform".StatusBalk4;
      =     L 0.0;
      BLD   103;
      A     "Geheugen.Platform".MoveBalk4;
      =     L 0.1;
      BLD   103;
      A     "Geheugen.Platform".StatusBalk2;
      =     L 0.2;
      BLD   103;
      A     "Geheugen.Platform".MoveBalk2;
      =     L 0.3;
      BLD   103;
      CALL  "Sub.Keuze.Sta.A.or.B" (
           Station                  := 0,
           StatusBalk1              := L 0.0,
           MoveBalk1                := L 0.1,
           StatusBalk2              := L 0.2,
           MoveBalk2                := L 0.3,
           huidige                  := "Stap 2.2",
           volgende                 := "Stap 2.4");
      NOP   0;
NETWORK
TITLE = Stap 2.2 -> Stap 3.2
//Naar Station B
      A     "Geheugen.Platform".StatusBalk2;
      =     L 0.0;
      BLD   103;
      A     "Geheugen.Platform".MoveBalk2;
      =     L 0.1;
      BLD   103;
      A     "Geheugen.Platform".StatusBalk4;
      =     L 0.2;
      BLD   103;
      A     "Geheugen.Platform".MoveBalk4;
      =     L 0.3;
      BLD   103;
      CALL  "Sub.Keuze.Sta.A.or.B" (
           Station                  := 1,
           StatusBalk1              := L 0.0,
           MoveBalk1                := L 0.1,
           StatusBalk2              := L 0.2,
           MoveBalk2                := L 0.3,
           huidige                  := "Stap 2.2",
           volgende                 := "Stap 3.2");
      NOP   0;
NETWORK
TITLE = Stap 2.2 -> Stap 3.6
//Station A + B
      A     "Geheugen.Platform".StatusBalk4;
      AN    "Geheugen.Platform".MoveBalk4;
      AN    "Geheugen.Platform".StatusBalk2;
      A     "Geheugen.Platform".MoveBalk2;
      =     L 0.0;
      BLD   103;
      CALL  "Sub.Basis" (
           voorwaarde               := L 0.0,
           huidige                  := "Stap 2.2",
           volgende                 := "Stap 3.6");
      NOP   0;
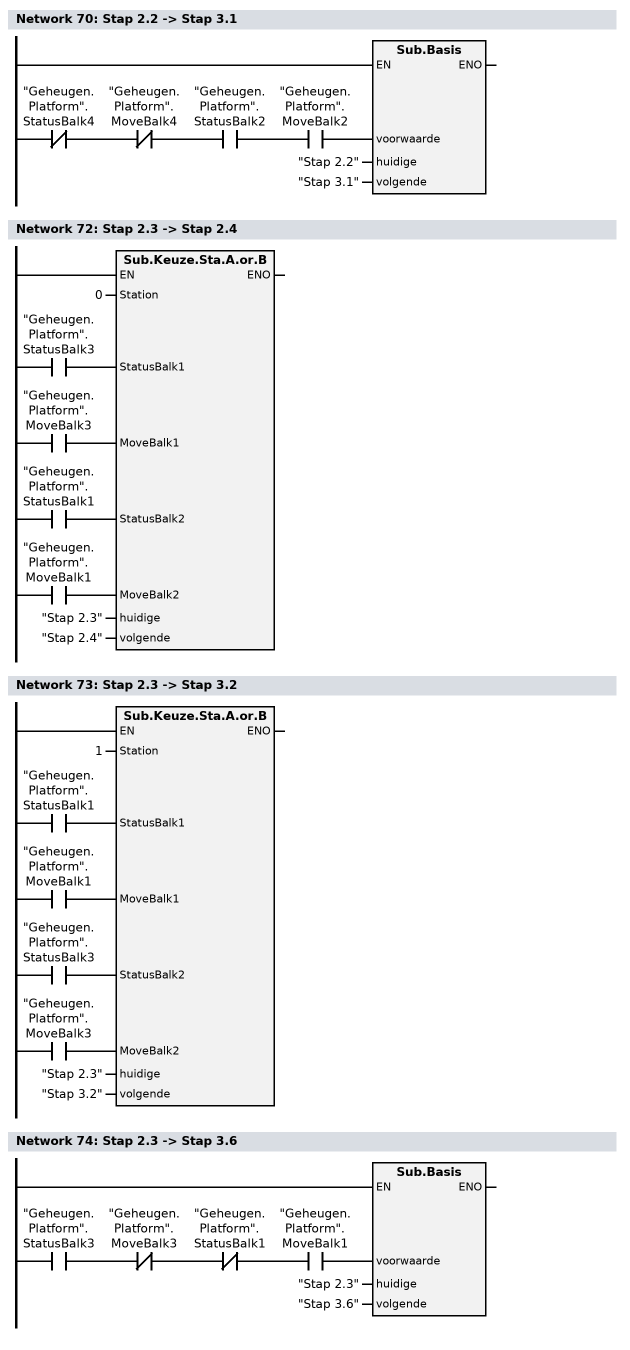
NETWORK
TITLE = Stap 2.2 -> Stap 3.1
//Geen actie
//
      AN    "Geheugen.Platform".StatusBalk4;
      AN    "Geheugen.Platform".MoveBalk4;
      A     "Geheugen.Platform".StatusBalk2;
      A     "Geheugen.Platform".MoveBalk2;
      =     L 0.0;
      BLD   103;
      CALL  "Sub.Basis" (
           voorwaarde               := L 0.0,
           huidige                  := "Stap 2.2",
           volgende                 := "Stap 3.1");
      NOP   0;
NETWORK
TITLE =
//*********************************************//
// Function: Einde Waarde Counter CO: 7        //
//           Begin Waarde Counter CO: 8        //
//*********************************************//
      NOP   0;
NETWORK
TITLE = Stap 2.3 -> Stap 2.4
//Naar Station A
      A     "Geheugen.Platform".StatusBalk3;
      =     L 0.0;
      BLD   103;
      A     "Geheugen.Platform".MoveBalk3;
      =     L 0.1;
      BLD   103;
      A     "Geheugen.Platform".StatusBalk1;
      =     L 0.2;
      BLD   103;
      A     "Geheugen.Platform".MoveBalk1;
      =     L 0.3;
      BLD   103;
      CALL  "Sub.Keuze.Sta.A.or.B" (
           Station                  := 0,
           StatusBalk1              := L 0.0,
           MoveBalk1                := L 0.1,
           StatusBalk2              := L 0.2,
           MoveBalk2                := L 0.3,
           huidige                  := "Stap 2.3",
           volgende                 := "Stap 2.4");
      NOP   0;
NETWORK
TITLE = Stap 2.3 -> Stap 3.2
//Naar Station B
      A     "Geheugen.Platform".StatusBalk1;
      =     L 0.0;
      BLD   103;
      A     "Geheugen.Platform".MoveBalk1;
      =     L 0.1;
      BLD   103;
      A     "Geheugen.Platform".StatusBalk3;
      =     L 0.2;
      BLD   103;
      A     "Geheugen.Platform".MoveBalk3;
      =     L 0.3;
      BLD   103;
      CALL  "Sub.Keuze.Sta.A.or.B" (
           Station                  := 1,
           StatusBalk1              := L 0.0,
           MoveBalk1                := L 0.1,
           StatusBalk2              := L 0.2,
           MoveBalk2                := L 0.3,
           huidige                  := "Stap 2.3",
           volgende                 := "Stap 3.2");
      NOP   0;
NETWORK
TITLE = Stap 2.3 -> Stap 3.6
//Station A + B
      A     "Geheugen.Platform".StatusBalk3;
      AN    "Geheugen.Platform".MoveBalk3;
      AN    "Geheugen.Platform".StatusBalk1;
      A     "Geheugen.Platform".MoveBalk1;
      =     L 0.0;
      BLD   103;
      CALL  "Sub.Basis" (
           voorwaarde               := L 0.0,
           huidige                  := "Stap 2.3",
           volgende                 := "Stap 3.6");
      NOP   0;
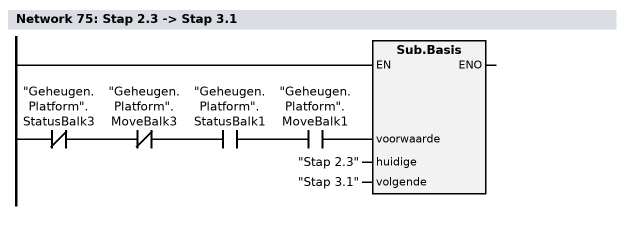
NETWORK
TITLE = Stap 2.3 -> Stap 3.1
//Geen actie
//
      AN    "Geheugen.Platform".StatusBalk3;
      AN    "Geheugen.Platform".MoveBalk3;
      A     "Geheugen.Platform".StatusBalk1;
      A     "Geheugen.Platform".MoveBalk1;
      =     L 0.0;
      BLD   103;
      CALL  "Sub.Basis" (
           voorwaarde               := L 0.0,
           huidige                  := "Stap 2.3",
           volgende                 := "Stap 3.1");
      NOP   0;
NETWORK
TITLE =
//*********************************************//
// Function: Einde Waarde Counter CO: 8        //
//           Begin Station Procédure           //
//*********************************************//
      NOP   0;
END_FUNCTION

FUNCTION "Simulatie" : VOID	// FC 6
VERSION : 0.1
BEGIN
// (block stored without names or comments; labels and parameter names are numbered)
END_FUNCTION

FUNCTION "Watch.Dog" : VOID	// FC 7
VERSION : 0.1
BEGIN
// (block stored without names or comments; labels and parameter names are numbered)
END_FUNCTION

FUNCTION "Sub.Basis" : VOID	// FC 14
VERSION : 0.1
VAR_INPUT
  voorwaarde : BOOL ;
END_VAR
VAR_IN_OUT
  huidige : BOOL ;
  volgende : BOOL ;
END_VAR
BEGIN
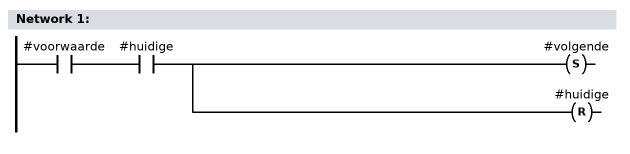
NETWORK
TITLE =
      A     #voorwaarde;
      A     #huidige;
      S     #volgende;
      R     #huidige;
END_FUNCTION

FUNCTION "Sub.Keuze" : VOID	// FC 15
VERSION : 0.1
VAR_INPUT
  BalkWaarde : INT ;
END_VAR
VAR_IN_OUT
  huidge : BOOL ;
  volgende : BOOL ;
END_VAR
BEGIN
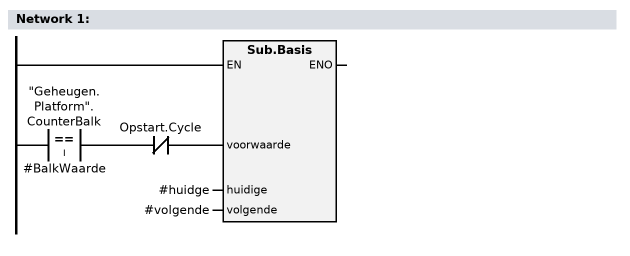
NETWORK
TITLE =
      A(;
      L     "Geheugen.Platform".CounterBalk;
      L     #BalkWaarde;
      ==I;
      );
      AN    "Opstart.Cycle";
      =     L 0.0;
      BLD   103;
      CALL  "Sub.Basis" (
           voorwaarde               := L 0.0,
           huidige                  := #huidge,
           volgende                 := #volgende);
      NOP   0;
END_FUNCTION

FUNCTION "Sub.Keuze.Sta.A.or.B" : VOID	// FC 16
VERSION : 0.1
VAR_INPUT
  Station : INT ;
  StatusBalk1 : BOOL ;
  MoveBalk1 : BOOL ;
  StatusBalk2 : BOOL ;
  MoveBalk2 : BOOL ;
END_VAR
VAR_IN_OUT
  huidige : BOOL ;
  volgende : BOOL ;
END_VAR
VAR_TEMP
  stationA : BOOL ;
  StationB : BOOL ;
END_VAR
BEGIN
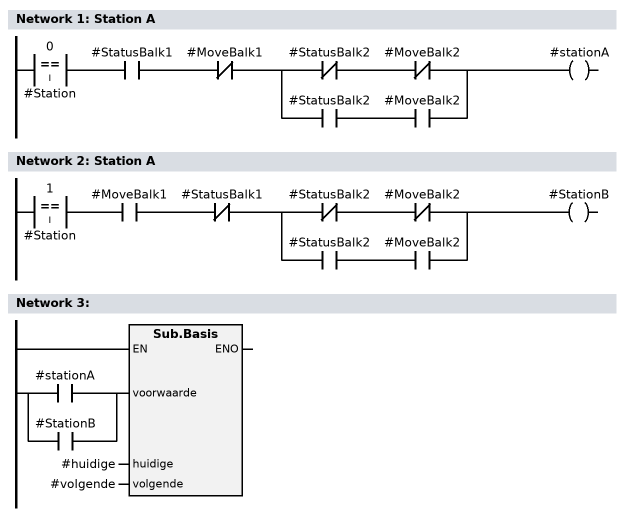
NETWORK
TITLE = Station A
      A(;
      L     0;
      L     #Station;
      ==I;
      );
      A     #StatusBalk1;
      AN    #MoveBalk1;
      A(;
      AN    #StatusBalk2;
      AN    #MoveBalk2;
      O;
      A     #StatusBalk2;
      A     #MoveBalk2;
      );
      =     #stationA;
NETWORK
TITLE = Station A
      A(;
      L     1;
      L     #Station;
      ==I;
      );
      A     #MoveBalk1;
      AN    #StatusBalk1;
      A(;
      AN    #StatusBalk2;
      AN    #MoveBalk2;
      O;
      A     #StatusBalk2;
      A     #MoveBalk2;
      );
      =     #StationB;
NETWORK
TITLE =
      A(;
      O     #stationA;
      O     #StationB;
      );
      =     L 1.0;
      BLD   103;
      CALL  "Sub.Basis" (
           voorwaarde               := L 1.0,
           huidige                  := #huidige,
           volgende                 := #volgende);
      NOP   0;
END_FUNCTION

DATA_BLOCK "Geheugen.Platform"	// DB 1
VERSION : 0.1
  STRUCT
   StatusBalk1 : BOOL ;
   StatusBalk2 : BOOL ;
   StatusBalk3 : BOOL ;
   StatusBalk4 : BOOL ;
   StatusBalk5 : BOOL ;
   StatusBalk6 : BOOL ;
   StatusBalk7 : BOOL ;
   StatusBalk8 : BOOL ;
   MoveBalk1 : BOOL ;
   MoveBalk2 : BOOL ;
   MoveBalk3 : BOOL ;
   MoveBalk4 : BOOL ;
   MoveBalk5 : BOOL ;
   MoveBalk6 : BOOL ;
   MoveBalk7 : BOOL ;
   MoveBalk8 : BOOL ;
   CounterBalk : INT ;
  END_STRUCT ;	
BEGIN
END_DATA_BLOCK

DATA_BLOCK "Geheugen.Instellingen"	// DB 2
VERSION : 0.1
  STRUCT
   FoutControle : BOOL ;
  END_STRUCT ;	
BEGIN
END_DATA_BLOCK

ORGANIZATION_BLOCK "Programma.Cyclus"	// OB 1
TITLE = "Main Program Sweep (Cycle)"
VERSION : 0.1
VAR_TEMP
  OB1_EV_CLASS : BYTE ;	//Bits 0-3 = 1 (Coming event), Bits 4-7 = 1 (Event class 1)
  OB1_SCAN_1 : BYTE ;	//1 (Cold restart scan 1 of OB 1), 3 (Scan 2-n of OB 1)
  OB1_PRIORITY : BYTE ;	//Priority of OB Execution
  OB1_OB_NUMBR : BYTE ;	//1 (Organization block 1, OB1)
  OB1_RESERVED_1 : BYTE ;	//Reserved for system
  OB1_RESERVED_2 : BYTE ;	//Reserved for system
  OB1_PREV_CYCLE : INT ;	//Cycle time of previous OB1 scan (milliseconds)
  OB1_MIN_CYCLE : INT ;	//Minimum cycle time of OB1 (milliseconds)
  OB1_MAX_CYCLE : INT ;	//Maximum cycle time of OB1 (milliseconds)
  OB1_DATE_TIME : DATE_AND_TIME ;	//Date and time OB1 started
END_VAR
BEGIN
NETWORK
TITLE =
      CALL  "Grafcet";
END_ORGANIZATION_BLOCK

ORGANIZATION_BLOCK "COMPLETE RESTART"	// OB 100
TITLE = "Complete Restart"
AUTHOR : B.Stijn
VERSION : 0.1
VAR_TEMP
  OB100_EV_CLASS : BYTE ;	//16#13, Event class 1, Entering event state, Event logged in diagnostic buffer
  OB100_STRTUP : BYTE ;	//16#81/82/83/84 Method of startup
  OB100_PRIORITY : BYTE ;	//Priority of OB Execution
  OB100_OB_NUMBR : BYTE ;	//100 (Organization block 100, OB100)
  OB100_RESERVED_1 : BYTE ;	//Reserved for system
  OB100_RESERVED_2 : BYTE ;	//Reserved for system
  OB100_STOP : WORD ;	//Event that caused CPU to stop (16#4xxx)
  OB100_STRT_INFO : DWORD ;	//Information on how system started
  OB100_DATE_TIME : DATE_AND_TIME ;	//Date and time OB100 started
END_VAR
BEGIN
NETWORK
TITLE = Opstart Merker
      AN    "Restart.OB100";
      S     "Restart.OB100";
NETWORK
TITLE = Resetten stappen
      L     0;
      T     MB 0;
      T     MB 1;
      T     MB 2;
      T     MB 3;
      T     MB 4;
      T     MB 5;
      NOP   0;
NETWORK
TITLE =
      AN    "Stap 0.0";
      S     "Stap 0.0";
END_ORGANIZATION_BLOCK

SYMBOL_TABLE
"I/O.Send"	FC 1	FC 1
"Noodstop.relais"	I 124.4	BOOL
"IB0"	MB 10	BYTE
"IB124"	MB 11	BYTE
"QB0"	MB 12	BYTE
"QB124"	MB 13	BYTE
"Programma.Cyclus"	OB 1	OB 1
END_SYMBOL_TABLE

FUNCTION "I/O.Send" : VOID	// FC 1
VERSION : 0.1
BEGIN
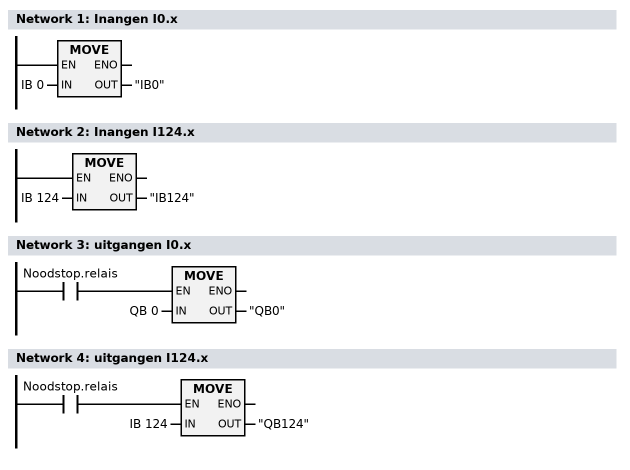
NETWORK
TITLE = Inangen I0.x
      L     IB 0;
      T     "IB0";
      NOP   0;
NETWORK
TITLE = Inangen I124.x
      L     IB 124;
      T     "IB124";
      NOP   0;
NETWORK
TITLE = uitgangen I0.x
      A     "Noodstop.relais";
      JNB   _001;
      L     QB 0;
      T     "QB0";
_001: NOP   0;
NETWORK
TITLE = uitgangen I124.x
      A     "Noodstop.relais";
      JNB   _002;
      L     IB 124;
      T     "QB124";
_002: NOP   0;
END_FUNCTION

ORGANIZATION_BLOCK "Programma.Cyclus"	// OB 1
TITLE = "Main Program Sweep (Cycle)"
VERSION : 0.1
VAR_TEMP
  OB1_EV_CLASS : BYTE ;	//Bits 0-3 = 1 (Coming event), Bits 4-7 = 1 (Event class 1)
  OB1_SCAN_1 : BYTE ;	//1 (Cold restart scan 1 of OB 1), 3 (Scan 2-n of OB 1)
  OB1_PRIORITY : BYTE ;	//Priority of OB Execution
  OB1_OB_NUMBR : BYTE ;	//1 (Organization block 1, OB1)
  OB1_RESERVED_1 : BYTE ;	//Reserved for system
  OB1_RESERVED_2 : BYTE ;	//Reserved for system
  OB1_PREV_CYCLE : INT ;	//Cycle time of previous OB1 scan (milliseconds)
  OB1_MIN_CYCLE : INT ;	//Minimum cycle time of OB1 (milliseconds)
  OB1_MAX_CYCLE : INT ;	//Maximum cycle time of OB1 (milliseconds)
  OB1_DATE_TIME : DATE_AND_TIME ;	//Date and time OB1 started
END_VAR
BEGIN
// (block stored without names or comments; labels and parameter names are numbered)
END_ORGANIZATION_BLOCK

SYMBOL_TABLE
"Productie_teller_Station"	C 0	COUNTER
"Productie_teller_Stat_A"	C 1	COUNTER
"Productie_teller_Stat_B"	C 2	COUNTER
"Productie_teller_In_Waar"	C 3	COUNTER
"SIM.Positie.Staven"	C 4	COUNTER
"Positionering.counter"	C 5	COUNTER
"SIM.OB1"	DB 2	DB 2	// Simualtie
"SIM.USERS"	DB 3	DB 3
"Positionering"	DB 4	DB 4
"Uitgangen Sturen"	FC 1	FC 1
"Timers + Counters"	FC 2	FC 2
"Grafcet Station A"	FC 3	FC 3
"Grafcet Station B"	FC 4	FC 4
"Simulatie_Run"	FC 5	FC 5
"Opstart_FC"	FC 6	FC 6
"Grafcet_Platform"	FC 7	FC 7	// Grafcet_Platform
"Ingang -> Merker"	FC 8	FC 8
"DB_Function"	FC 9	FC 9
"SIM.OB100"	FC 10	FC 10
"SIM.user"	FC 11	FC 11
"Positionering_balken"	FC 12	FC 12
"Sub_routine"	FC 14	FC 14
"Opstart_subroutine"	FC 15	FC 15
"Sub_routine_gelijk"	FC 16	FC 16
"Sub_route_Station_samen"	FC 17	FC 17
"SIM.SUBR.Y-As"	FC 19	FC 19
"SIM.LOGIN"	FC 20	FC 20
"SIM.Move.X-As"	FC 21	FC 21
"SIM.BALK.Reset"	FC 22	FC 22
"SUB.Posit"	FC 23	FC 23
"Stap 0.0"	M 0.0	BOOL
"Stap 0.1"	M 0.1	BOOL
"Stap 0.2"	M 0.2	BOOL
"Stap 0.3"	M 0.3	BOOL
"Stap 0.4"	M 0.4	BOOL
"Stap 0.5"	M 0.5	BOOL
"Stap 1.1"	M 1.1	BOOL
"Stap 1.2"	M 1.2	BOOL
"Stap 1.3"	M 1.3	BOOL
"Stap 1.4"	M 1.4	BOOL
"Stap 1.5"	M 1.5	BOOL
"Stap 2.0"	M 2.0	BOOL
"Stap 2.1"	M 2.1	BOOL
"Stap 2.2"	M 2.2	BOOL
"Stap 2.3"	M 2.3	BOOL
"Stap 2.4"	M 2.4	BOOL
"Stap 2.5"	M 2.5	BOOL
"Start"	M 5.0	BOOL
"Stop"	M 5.1	BOOL
"Piston A in"	M 5.2	BOOL
"Piston A uit"	M 5.3	BOOL
"Piston A onder"	M 5.4	BOOL
"Piston A boven"	M 5.5	BOOL
"Piston B in"	M 5.6	BOOL
"Piston B uit"	M 5.7	BOOL
"Piston B onder"	M 6.0	BOOL
"Piston B boven"	M 6.1	BOOL
"Proxi Pos 1"	M 6.2	BOOL
"Proxi Pos 2"	M 6.3	BOOL
"Motor Rechts"	M 7.1	BOOL
"Piston A Op-Neer"	M 7.2	BOOL
"Piston A Uit-In"	M 7.3	BOOL
"Piston B Op-Neer"	M 7.4	BOOL
"Piston B Uit-In"	M 7.5	BOOL
"Sign.Rood"	M 7.6	BOOL
"Sign.Groen"	M 7.7	BOOL
"Motor Links"	M 8.0	BOOL
"Opstart"	M 10.0	BOOL
"SIM.reset.C4"	M 10.1	BOOL
"P.M10.2"	M 10.2	BOOL
"SIM.opstart.5S"	M 10.3	BOOL
"admin"	M 11.0	BOOL
"monitor"	M 11.1	BOOL
"operate"	M 11.2	BOOL
"user"	M 11.3	BOOL
"SIM.User.Login"	M 11.4	BOOL
"SIM.User.logout"	M 11.5	BOOL
"SIM.USER.ERROR"	M 11.6	BOOL
"Sim.Start.Postitionering"	M 24.0	BOOL
"Postitionering.Station.A"	M 24.1	BOOL
"Postitionering.Station.B"	M 24.2	BOOL
"Postitionering.Return"	M 24.3	BOOL
"SIM.Positie.Save"	M 24.4	BOOL
"SIM.Positie.Zoom"	M 24.5	BOOL
"Positionering.Stop"	M 24.6	BOOL
"Balk1"	M 25.0	BOOL
"Blak2"	M 25.1	BOOL
"Balk3"	M 25.2	BOOL
"Balk4"	M 25.3	BOOL
"Balk5"	M 25.4	BOOL
"Balk6"	M 25.5	BOOL
"Balk7"	M 25.6	BOOL
"Balk8"	M 25.7	BOOL
"Test Piston A"	M 30.0	BOOL
"Fout Controle station A"	M 30.1	BOOL
"Fout Reset station A"	M 30.2	BOOL
"Test station B"	M 30.3	BOOL
"Fout Controle station B"	M 30.4	BOOL
"Fout_Motor"	M 30.5	BOOL
"Foint Station_A_B"	M 30.6	BOOL
"Stop Meker"	M 30.7	BOOL
"DBW0 == DBW2"	M 31.0	BOOL
"DBW0 < DBW2"	M 31.1	BOOL
"DBW0 != 0"	M 31.2	BOOL
"SIM.Start.StaA"	M 31.3	BOOL
"SIM.Start.StaB"	M 31.4	BOOL
"SIM.Start"	M 31.5	BOOL
"SIM.Stop"	M 31.6	BOOL
"DBW0 == 0"	M 32.0	BOOL
"INI.Stations"	M 33.0	BOOL
"Start Stat A + B"	M 33.1	BOOL
"Blinker 5s"	M 100.5	BOOL
"Restart"	M 101.1	BOOL
"Ingangen 0.x"	MB 5	BYTE
"Ingangen 124.x"	MB 6	BYTE
"Uitgangen 0.x"	MB 7	BYTE
"Uitgangen 124.x"	MB 8	BYTE
"Positie.balken"	MB 25	BYTE
"SIM.C.Positie.BCD"	MW 12	WORD	// Balk die zich bevind voor de sensoren(bcd waarde)
"SIM.C.Positie.INT"	MW 14	INT	// Balk die zich bevind voor de sensoren(int waarde)
"SIM.C.Postie.Stat.A"	MW 16	INT	// Balk die zich bevind voor station A
"SIM.C.Postie.Stat.B"	MW 18	INT	// Balk due zich bevind voor station B
"SIM.Station.A"	MW 20	WORD
"SIM.Station.B"	MW 22	WORD
"COMPLETE RESTART"	OB 100	OB 100	// Complete Restart
"Motor controler"	T 0	TIMER
"Timer Contr Neer A"	T 1	TIMER
"Timer contr uit A"	T 2	TIMER
"Timer contr uit B"	T 3	TIMER
"Timer contr neer B"	T 4	TIMER
"Hori Station B"	T 5	TIMER
"Verti Station B"	T 6	TIMER
"SIM.SUBR.T1"	T 7	TIMER
"SIM.SUBR.T2"	T 8	TIMER
"SIM.User.Error.T"	T 9	TIMER
"Vertraging.Station.off"	T 10	TIMER
"Vertraging.Station.Aan"	T 11	TIMER
END_SYMBOL_TABLE

FUNCTION "Uitgangen Sturen" : VOID	// FC 1
VERSION : 0.1
BEGIN
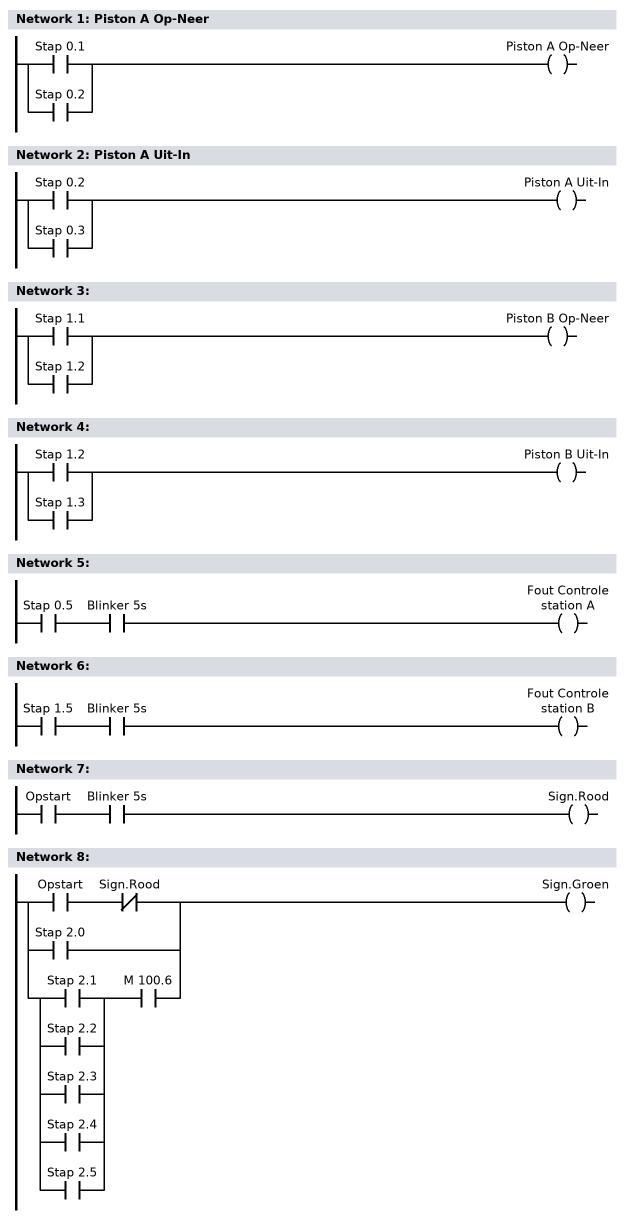
NETWORK
TITLE = Piston A Op-Neer
      O     "Stap 0.1";
      O     "Stap 0.2";
      =     "Piston A Op-Neer";
NETWORK
TITLE = Piston A Uit-In
      O     "Stap 0.2";
      O     "Stap 0.3";
      =     "Piston A Uit-In";
NETWORK
TITLE =
      O     "Stap 1.1";
      O     "Stap 1.2";
      =     "Piston B Op-Neer";
NETWORK
TITLE =
      O     "Stap 1.2";
      O     "Stap 1.3";
      =     "Piston B Uit-In";
NETWORK
TITLE =
      A     "Stap 0.5";
      A     "Blinker 5s";
      =     "Fout Controle station A";
NETWORK
TITLE =
      A     "Stap 1.5";
      A     "Blinker 5s";
      =     "Fout Controle station B";
NETWORK
TITLE =
      A     "Opstart";
      A     "Blinker 5s";
      =     "Sign.Rood";
NETWORK
TITLE =
      A     "Opstart";
      AN    "Sign.Rood";
      O     "Stap 2.0";
      O;
      A(;
      O     "Stap 2.1";
      O     "Stap 2.2";
      O     "Stap 2.3";
      O     "Stap 2.4";
      O     "Stap 2.5";
      );
      A     M 100.6;
      =     "Sign.Groen";
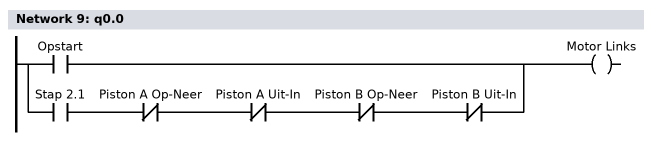
NETWORK
TITLE = q0.0
      O     "Opstart";
      O;
      A     "Stap 2.1";
      AN    "Piston A Op-Neer";
      AN    "Piston A Uit-In";
      AN    "Piston B Op-Neer";
      AN    "Piston B Uit-In";
      =     "Motor Links";
END_FUNCTION

FUNCTION "Timers + Counters" : VOID	// FC 2
VERSION : 0.1
BEGIN
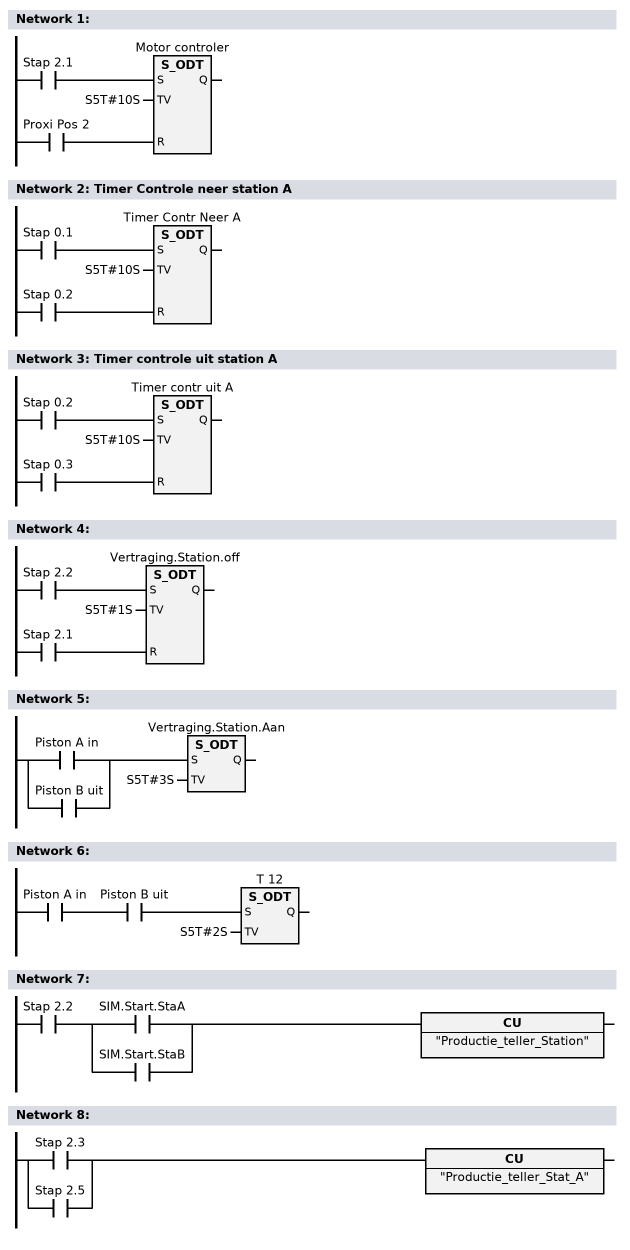
NETWORK
TITLE =
      A     "Stap 2.1";
      L     S5T#10S;
      SD    "Motor controler";
      A     "Proxi Pos 2";
      R     "Motor controler";
      NOP   0;
      NOP   0;
      NOP   0;
NETWORK
TITLE = Timer Controle neer station A
      A     "Stap 0.1";
      L     S5T#10S;
      SD    "Timer Contr Neer A";
      A     "Stap 0.2";
      R     "Timer Contr Neer A";
      NOP   0;
      NOP   0;
      NOP   0;
NETWORK
TITLE = Timer controle uit station A
      A     "Stap 0.2";
      L     S5T#10S;
      SD    "Timer contr uit A";
      A     "Stap 0.3";
      R     "Timer contr uit A";
      NOP   0;
      NOP   0;
      NOP   0;
NETWORK
TITLE =
      A     "Stap 2.2";
      L     S5T#1S;
      SD    "Vertraging.Station.off";
      A     "Stap 2.1";
      R     "Vertraging.Station.off";
      NOP   0;
      NOP   0;
      NOP   0;
NETWORK
TITLE =
      A(;
      O     "Piston A in";
      O     "Piston B uit";
      );
      L     S5T#3S;
      SD    "Vertraging.Station.Aan";
      NOP   0;
      NOP   0;
      NOP   0;
      NOP   0;
NETWORK
TITLE =
      A     "Piston A in";
      A     "Piston B uit";
      L     S5T#2S;
      SD    T 12;
      NOP   0;
      NOP   0;
      NOP   0;
      NOP   0;
NETWORK
TITLE =
      A     "Stap 2.2";
      A(;
      O     "SIM.Start.StaA";
      O     "SIM.Start.StaB";
      );
      CU    "Productie_teller_Station";
      BLD   101;
      NOP   0;
      NOP   0;
      NOP   0;
      NOP   0;
      NOP   0;
      NOP   0;
NETWORK
TITLE =
      A(;
      O     "Stap 2.3";
      O     "Stap 2.5";
      );
      CU    "Productie_teller_Stat_A";
      BLD   101;
      NOP   0;
      NOP   0;
      NOP   0;
      NOP   0;
      NOP   0;
      NOP   0;
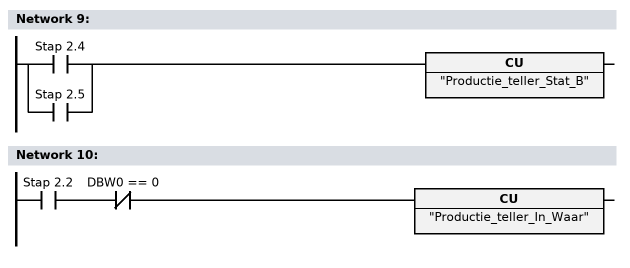
NETWORK
TITLE =
      A(;
      O     "Stap 2.4";
      O     "Stap 2.5";
      );
      CU    "Productie_teller_Stat_B";
      BLD   101;
      NOP   0;
      NOP   0;
      NOP   0;
      NOP   0;
      NOP   0;
      NOP   0;
NETWORK
TITLE =
      A     "Stap 2.2";
      AN    "DBW0 == 0";
      CU    "Productie_teller_In_Waar";
      BLD   101;
      NOP   0;
      NOP   0;
      NOP   0;
      NOP   0;
      NOP   0;
      NOP   0;
END_FUNCTION

FUNCTION "Grafcet Station A" : VOID	// FC 3
VERSION : 0.1
BEGIN
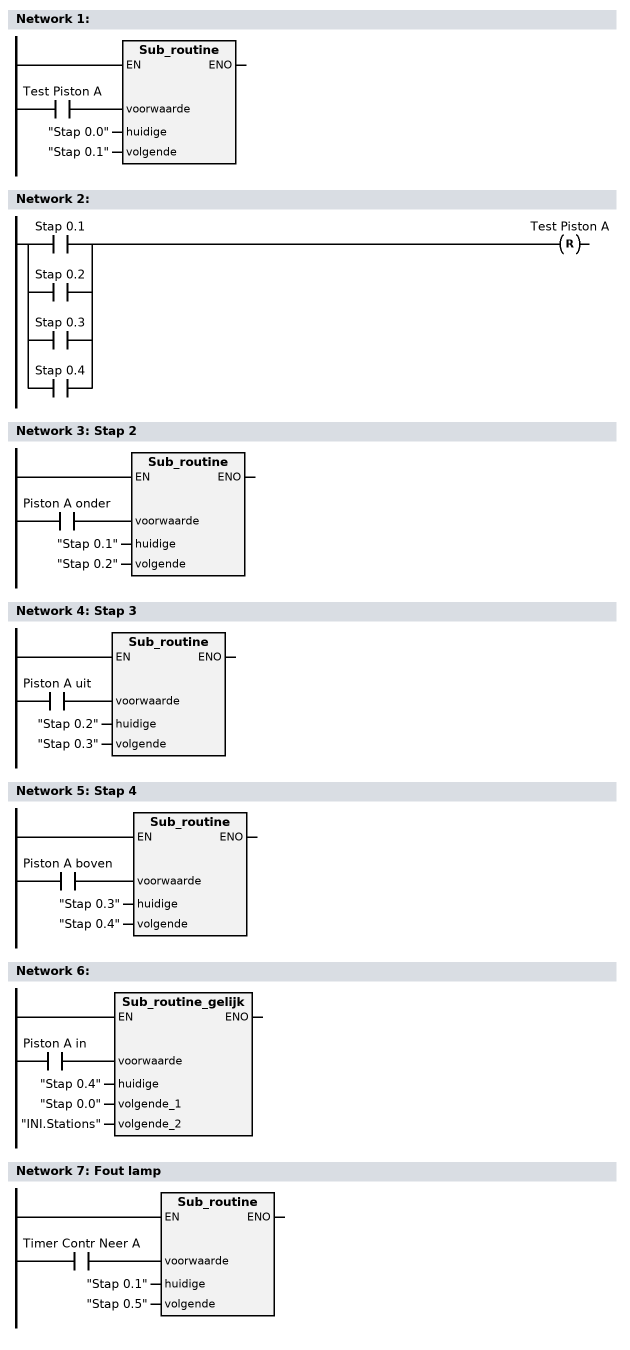
NETWORK
TITLE =
      A     "Test Piston A";
      =     L 0.0;
      BLD   103;
      CALL  "Sub_routine" (
           voorwaarde               := L 0.0,
           huidige                  := "Stap 0.0",
           volgende                 := "Stap 0.1");
      NOP   0;
NETWORK
TITLE =
      O     "Stap 0.1";
      O     "Stap 0.2";
      O     "Stap 0.3";
      O     "Stap 0.4";
      R     "Test Piston A";
NETWORK
TITLE = Stap 2
      A     "Piston A onder";
      =     L 0.0;
      BLD   103;
      CALL  "Sub_routine" (
           voorwaarde               := L 0.0,
           huidige                  := "Stap 0.1",
           volgende                 := "Stap 0.2");
      NOP   0;
NETWORK
TITLE = Stap 3
      A     "Piston A uit";
      =     L 0.0;
      BLD   103;
      CALL  "Sub_routine" (
           voorwaarde               := L 0.0,
           huidige                  := "Stap 0.2",
           volgende                 := "Stap 0.3");
      NOP   0;
NETWORK
TITLE = Stap 4
      A     "Piston A boven";
      =     L 0.0;
      BLD   103;
      CALL  "Sub_routine" (
           voorwaarde               := L 0.0,
           huidige                  := "Stap 0.3",
           volgende                 := "Stap 0.4");
      NOP   0;
NETWORK
TITLE =
      A     "Piston A in";
      =     L 0.0;
      BLD   103;
      CALL  "Sub_routine_gelijk" (
           voorwaarde               := L 0.0,
           huidige                  := "Stap 0.4",
           volgende_1               := "Stap 0.0",
           volgende_2               := "INI.Stations");
      NOP   0;
NETWORK
TITLE = Fout lamp
      A     "Timer Contr Neer A";
      =     L 0.0;
      BLD   103;
      CALL  "Sub_routine" (
           voorwaarde               := L 0.0,
           huidige                  := "Stap 0.1",
           volgende                 := "Stap 0.5");
      NOP   0;
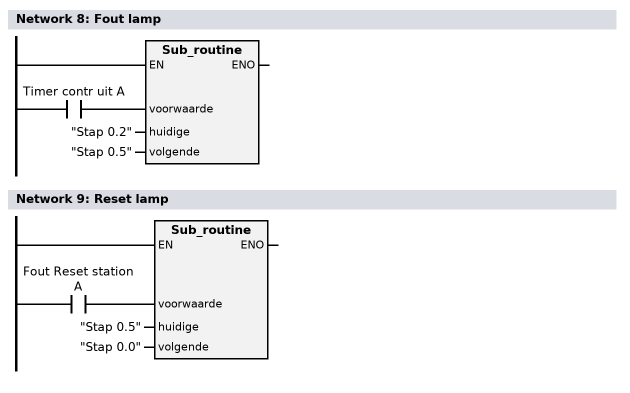
NETWORK
TITLE = Fout lamp
      A     "Timer contr uit A";
      =     L 0.0;
      BLD   103;
      CALL  "Sub_routine" (
           voorwaarde               := L 0.0,
           huidige                  := "Stap 0.2",
           volgende                 := "Stap 0.5");
      NOP   0;
NETWORK
TITLE = Reset lamp
      A     "Fout Reset station A";
      =     L 0.0;
      BLD   103;
      CALL  "Sub_routine" (
           voorwaarde               := L 0.0,
           huidige                  := "Stap 0.5",
           volgende                 := "Stap 0.0");
      NOP   0;
END_FUNCTION

FUNCTION "Grafcet Station B" : VOID	// FC 4
VERSION : 0.1
BEGIN
